KUKA KRL program: EPS_2_25252_SD5_A_20250910061729.src

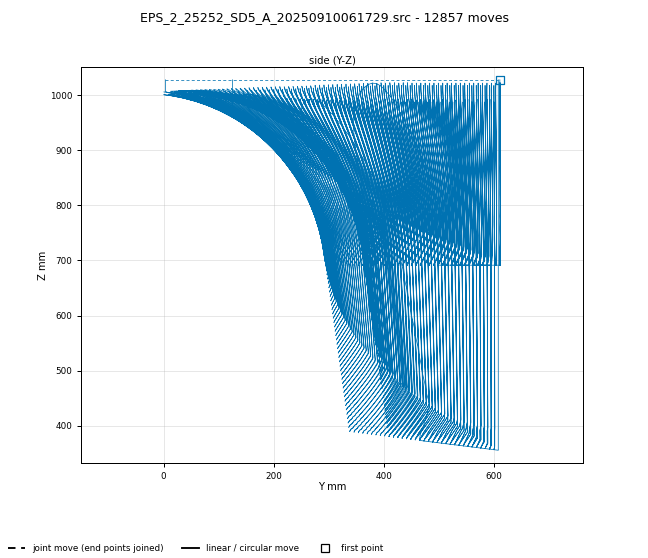
[picture p0: tool path of EPS_2_25252_SD5_A_20250910061729.src, 12857 of 12859 moves have a stored position in this frame; points joined in program order, loops and branches not executed]
&ACCESS RVP
&REL 4
&COMMENT QRS 19112012
&PARAM EDITMASK = *
DEF PART()
EXT BAS (BAS_COMMAND :IN,REAL :IN )
INT I
BAS (#INITMOV,0 )

;KUKA QRS Post kuka4.cps  Date:22-06-2017 !

File_ID=2833

QRS_PRE_INIT()

;Init var - Until changes are made in qrs_pre_init
Outlet_Square_prg=0
Inlet_1_Square_prg=0
Inlet_2_Square_prg=0
Inlet_3_Square_prg=0
Inlet_4_Square_prg=0
Inlet_5_Square_prg=0

Outlet_1={X 0.000, Y 400.000, Z 713.000, B 0.000, E1 0.000 }
Inlet_1={X 0.000, Y 400.000, Z 683.000, B 0.000, E1 212.000 }
Outlet_1_type=610
Inlet_1_type=610
;QRS#1=Sidecore dimensions
;QRS#2=600-24" Concrete
;QRS#3=600-24" Concrete
;QRS#4=
;QRS#5=
;QRS#6=
;QRS#7=
;QRS#8=
;QRS#9=S306-34L
;QRS#10=S306-34L
;QRS#11=
;QRS#12=
;QRS#13=
;QRS#14=
;QRS#15=
;QRS#16=1220x127x1372 4,5'
;QRS#17=EPS Height
;QRS#18=1018
;QRS#19=*
;QRS#20= UPDATED VERSION 22-06-2017
;QRS#21=*
Outlet_Square=0450
Inlet_1_Square=0450
Inlet_2_Square=0
Inlet_3_Square=0
Inlet_4_Square=0
Inlet_5_Square=0
Mill_Square=1
Outlet_Square_Prg=264
Inlet_1_Square_prg=264

QRS_INIT()

$ADVANCE=5

; T1
PTP {E1 178.273,E2 178.273}
PTP {X 0,Y 610.751,A -85,B 0,C 180,E1 178.273,E2 178.273,E3 0,E4 0,E5 0,E6 0}
QRS_SPEED_INIT()
LIN {X 0,Y 610.751,Z 1028,A -85,B 0,C 180,E1 178.273,E2 178.273,E3 0,E4 0,E5 0,E6 0} C_VEL
LIN {X 0,Y 610.751,Z 693.44,A -85,B 0,C 180,E1 178.273,E2 178.273} C_VEL
LIN {X 0,Y 610.777,Z 691.44,A -85,B 0,C 180,E1 178.46,E2 178.46} C_VEL
LIN {X 0,Y 611.879,Z 691.44,A -85,B 0,C 180,E1 181.167,E2 181.167} C_VEL
LIN {X 0,Y 611.804,Z 691.44,A -85,B 0,C 180,E1 188.197,E2 188.197} C_VEL
LIN {X 0,Y 611.819,Z 691.44,A -85,B 0,C 180,E1 195.354,E2 195.354} C_VEL
LIN {X 0,Y 611.767,Z 691.44,A -85,B 0,C 180,E1 202.769,E2 202.769} C_VEL
LIN {X 0,Y 611.74,Z 691.44,A -85,B 0,C 180,E1 210.614,E2 210.614} C_VEL
LIN {X 0,Y 610.579,Z 691.44,A -85,B 0,C 180,E1 217.262,E2 217.262} C_VEL
LIN {X 0,Y 611.716,Z 691.44,A -85,B 0,C 180,E1 219.161,E2 219.161} C_VEL
LIN {X 0,Y 610.312,Z 691.44,A -85,B 0,C 180,E1 222.361,E2 222.361} C_VEL
LIN {X 0,Y 610.625,Z 691.44,A -85,B 0,C 180,E1 225.583,E2 225.583} C_VEL
LIN {X 0,Y 611.712,Z 691.44,A -85,B 0,C 180,E1 227.764,E2 227.764} C_VEL
LIN {X 0,Y 611.693,Z 691.44,A -85,B 0,C 180,E1 235.933,E2 235.933} C_VEL
LIN {X 0,Y 611.734,Z 691.44,A -85,B 0,C 180,E1 236.287,E2 236.287} C_VEL
LIN {X 0,Y 611.056,Z 691.44,A -85,B 0,C 180,E1 236.42,E2 236.42} C_VEL
LIN {X 0,Y 610.433,Z 691.484,A -85,B 0,C 180,E1 236.481,E2 236.481} C_VEL
LIN {X 0,Y 611.412,Z 730.58,A -85,B 0,C 180,E1 237.083,E2 237.083} C_VEL
LIN {X 0,Y 611.517,Z 745.271,A -85,B 0,C 180,E1 237.336,E2 237.336} C_VEL
LIN {X 0,Y 611.325,Z 761.355,A -85,B 0,C 180,E1 237.681,E2 237.681} C_VEL
LIN {X 0,Y 611.672,Z 775.492,A -85,B 0,C 180,E1 238.087,E2 238.087} C_VEL
LIN {X 0,Y 611.736,Z 790.247,A -85,B 0,C 180,E1 238.57,E2 238.57} C_VEL
LIN {X 0,Y 611.693,Z 805.404,A -85,B 0,C 180,E1 239.145,E2 239.145} C_VEL
LIN {X 0,Y 611.448,Z 819.865,A -85,B 0,C 180,E1 239.763,E2 239.763} C_VEL
LIN {X 0,Y 611.625,Z 833.379,A -85,B 0,C 180,E1 240.435,E2 240.435} C_VEL
LIN {X 0,Y 611.599,Z 846.987,A -85,B 0,C 180,E1 241.179,E2 241.179} C_VEL
LIN {X 0,Y 611.634,Z 859.681,A -85,B 0,C 180,E1 241.947,E2 241.947} C_VEL
LIN {X 0,Y 611.641,Z 873.336,A -85,B 0,C 180,E1 242.859,E2 242.859} C_VEL
LIN {X 0,Y 611.572,Z 885.151,A -85,B 0,C 180,E1 243.716,E2 243.716} C_VEL
LIN {X 0,Y 611.333,Z 897.156,A -85,B 0,C 180,E1 244.659,E2 244.659} C_VEL
LIN {X 0,Y 611.276,Z 908.946,A -85,B 0,C 180,E1 245.678,E2 245.678} C_VEL
LIN {X 0,Y 611.472,Z 919.358,A -85,B 0,C 180,E1 246.662,E2 246.662} C_VEL
LIN {X 0,Y 611.734,Z 929.985,A -85,B 0,C 180,E1 247.752,E2 247.752} C_VEL
LIN {X 0,Y 611.445,Z 939.604,A -85,B 0,C 180,E1 248.799,E2 248.799} C_VEL
LIN {X 0,Y 611.088,Z 948.773,A -85,B 0,C 180,E1 249.876,E2 249.876} C_VEL
LIN {X 0,Y 611.074,Z 958.33,A -85,B 0,C 180,E1 251.115,E2 251.115} C_VEL
LIN {X 0,Y 611.399,Z 966.016,A -85,B 0,C 180,E1 252.202,E2 252.202} C_VEL
LIN {X 0,Y 611.821,Z 973.294,A -85,B 0,C 180,E1 253.324,E2 253.324} C_VEL
LIN {X 0,Y 611.107,Z 982.504,A -85,B 0,C 180,E1 254.862,E2 254.862} C_VEL
LIN {X 0,Y 610.739,Z 989.282,A -85,B 0,C 180,E1 256.129,E2 256.129} C_VEL
LIN {X 0,Y 610.875,Z 995.064,A -85,B 0,C 180,E1 257.336,E2 257.336} C_VEL
LIN {X 0,Y 611.566,Z 1001.374,A -85,B 0,C 180,E1 258.842,E2 258.842} C_VEL
LIN {X 0,Y 611.85,Z 1003.593,A -85,B 0,C 180,E1 259.441,E2 259.441} C_VEL
LIN {X 0,Y 611.525,Z 1005.813,A -85,B 0,C 180,E1 260.028,E2 260.028} C_VEL
LIN {X 0,Y 610.929,Z 1009.654,A -85,B 0,C 180,E1 261.203,E2 261.203} C_VEL
LIN {X 0,Y 610.672,Z 1012.99,A -85,B 0,C 180,E1 262.381,E2 262.381} C_VEL
LIN {X 0,Y 610.672,Z 1014.551,A -85,B 0,C 180,E1 262.97,E2 262.97} C_VEL
LIN {X 0,Y 611.06,Z 1017.122,A -85,B 0,C 180,E1 264.15,E2 264.15} C_VEL
LIN {X 0,Y 611.711,Z 1019.175,A -85,B 0,C 180,E1 265.329,E2 265.329} C_VEL
LIN {X 0,Y 611.37,Z 1020.807,A -85,B 0,C 180,E1 266.497,E2 266.497} C_VEL
LIN {X 0,Y 610.858,Z 1021.972,A -85,B 0,C 180,E1 267.634,E2 267.634} C_VEL
LIN {X 0,Y 610.688,Z 1022.778,A -85,B 0,C 180,E1 269.07,E2 269.07} C_VEL
LIN {X 0,Y 611.538,Z 1022.689,A -85,B 0,C 180,E1 271.17,E2 271.17} C_VEL
LIN {X 0,Y 611.319,Z 1021.671,A -85,B 0,C 180,E1 272.765,E2 272.765} C_VEL
LIN {X 0,Y 611.035,Z 1020.812,A -85,B 0,C 180,E1 273.51,E2 273.51} C_VEL
LIN {X 0,Y 610.805,Z 1019.195,A -85,B 0,C 180,E1 274.683,E2 274.683} C_VEL
LIN {X 0,Y 611.004,Z 1017.112,A -85,B 0,C 180,E1 275.855,E2 275.855} C_VEL
LIN {X 0,Y 611.55,Z 1014.528,A -85,B 0,C 180,E1 277.025,E2 277.025} C_VEL
LIN {X 0,Y 611.873,Z 1012.96,A -85,B 0,C 180,E1 277.609,E2 277.609} C_VEL
LIN {X 0,Y 611.24,Z 1009.637,A -85,B 0,C 180,E1 278.797,E2 278.797} C_VEL
LIN {X 0,Y 610.738,Z 1005.794,A -85,B 0,C 180,E1 279.99,E2 279.99} C_VEL
LIN {X 0,Y 610.738,Z 1000.148,A -85,B 0,C 180,E1 281.477,E2 281.477} C_VEL
LIN {X 0,Y 611.199,Z 995.041,A -85,B 0,C 180,E1 282.663,E2 282.663} C_VEL
LIN {X 0,Y 611.828,Z 989.347,A -85,B 0,C 180,E1 283.832,E2 283.832} C_VEL
LIN {X 0,Y 611.263,Z 982.265,A -85,B 0,C 180,E1 285.179,E2 285.179} C_VEL
LIN {X 0,Y 610.874,Z 973.74,A -85,B 0,C 180,E1 286.634,E2 286.634} C_VEL
LIN {X 0,Y 611.107,Z 964.917,A -85,B 0,C 180,E1 287.966,E2 287.966} C_VEL
LIN {X 0,Y 611.627,Z 956.005,A -85,B 0,C 180,E1 289.182,E2 289.182} C_VEL
LIN {X 0,Y 611.763,Z 951.156,A -85,B 0,C 180,E1 289.796,E2 289.796} C_VEL
LIN {X 0,Y 611.529,Z 944.982,A -85,B 0,C 180,E1 290.565,E2 290.565} C_VEL
LIN {X 0,Y 611.268,Z 937.362,A -85,B 0,C 180,E1 291.465,E2 291.465} C_VEL
LIN {X 0,Y 611.182,Z 926.924,A -85,B 0,C 180,E1 292.59,E2 292.59} C_VEL
LIN {X 0,Y 611.438,Z 916.307,A -85,B 0,C 180,E1 293.633,E2 293.633} C_VEL
LIN {X 0,Y 611.68,Z 905.115,A -85,B 0,C 180,E1 294.645,E2 294.645} C_VEL
LIN {X 0,Y 611.642,Z 894.627,A -85,B 0,C 180,E1 295.535,E2 295.535} C_VEL
LIN {X 0,Y 611.47,Z 882.904,A -85,B 0,C 180,E1 296.459,E2 296.459} C_VEL
LIN {X 0,Y 611.456,Z 869.528,A -85,B 0,C 180,E1 297.413,E2 297.413} C_VEL
LIN {X 0,Y 611.583,Z 857.645,A -85,B 0,C 180,E1 298.184,E2 298.184} C_VEL
LIN {X 0,Y 611.506,Z 843.831,A -85,B 0,C 180,E1 299.006,E2 299.006} C_VEL
LIN {X 0,Y 611.705,Z 829.667,A -85,B 0,C 180,E1 299.75,E2 299.75} C_VEL
LIN {X 0,Y 611.695,Z 816.022,A -85,B 0,C 180,E1 300.401,E2 300.401} C_VEL
LIN {X 0,Y 611.697,Z 800.989,A -85,B 0,C 180,E1 301.031,E2 301.031} C_VEL
LIN {X 0,Y 611.541,Z 786.837,A -85,B 0,C 180,E1 301.558,E2 301.558} C_VEL
LIN {X 0,Y 611.397,Z 780.445,A -85,B 0,C 180,E1 301.77,E2 301.77} C_VEL
LIN {X 0,Y 611.662,Z 771.874,A -85,B 0,C 180,E1 302.018,E2 302.018} C_VEL
LIN {X 0,Y 611.795,Z 756.357,A -85,B 0,C 180,E1 302.41,E2 302.41} C_VEL
LIN {X 0,Y 611.777,Z 742.708,A -85,B 0,C 180,E1 302.698,E2 302.698} C_VEL
LIN {X 0,Y 611.541,Z 723.406,A -85,B 0,C 180,E1 303.011,E2 303.011} C_VEL
LIN {X 0,Y 610.652,Z 696.32,A -85,B 0,C 180,E1 303.438,E2 303.438} C_VEL
LIN {X 0,Y 610.425,Z 691.44,A -85,B 0,C 180,E1 303.52,E2 303.52} C_VEL
LIN {X 0,Y 610.949,Z 691.44,A -85,B 0,C 180,E1 303.571,E2 303.571} C_VEL
LIN {X 0,Y 611.627,Z 691.44,A -85,B 0,C 180,E1 303.682,E2 303.682} C_VEL
LIN {X 0,Y 611.854,Z 691.44,A -85,B 0,C 180,E1 303.975,E2 303.975} C_VEL
LIN {X 0,Y 611.819,Z 691.44,A -85,B 0,C 180,E1 306.206,E2 306.206} C_VEL
LIN {X 0,Y 610.447,Z 691.44,A -85,B 0,C 180,E1 309.26,E2 309.26} C_VEL
LIN {X 0,Y 610.689,Z 691.44,A -85,B 0,C 180,E1 312.33,E2 312.33} C_VEL
LIN {X 0,Y 611.706,Z 691.44,A -85,B 0,C 180,E1 314.52,E2 314.52} C_VEL
LIN {X 0,Y 611.667,Z 691.44,A -85,B 0,C 180,E1 322.613,E2 322.613} C_VEL
LIN {X 0,Y 611.137,Z 691.44,A -85,B 0,C 180,E1 323.749,E2 323.749} C_VEL
LIN {X 0,Y 611.64,Z 691.44,A -85,B 0,C 180,E1 331.173,E2 331.173} C_VEL
LIN {X 0,Y 611.418,Z 691.44,A -85,B 0,C 180,E1 332.046,E2 332.046} C_VEL
LIN {X 0,Y 611.836,Z 691.44,A -85,B 0,C 180,E1 339.742,E2 339.742} C_VEL
LIN {X 0,Y 611.807,Z 691.44,A -85,B 0,C 180,E1 347.053,E2 347.053} C_VEL
LIN {X 0,Y 611.862,Z 691.44,A -85,B 0,C 180,E1 354.155,E2 354.155} C_VEL
LIN {X 0,Y 611.865,Z 691.44,A -85,B 0,C 180,E1 361.167,E2 361.167} C_VEL
LIN {X 0,Y 611.872,Z 691.44,A -85,B 0,C 180,E1 368.196,E2 368.196} C_VEL
LIN {X 0,Y 611.844,Z 691.44,A -85,B 0,C 180,E1 375.353,E2 375.353} C_VEL
LIN {X 0,Y 611.848,Z 691.44,A -85,B 0,C 180,E1 384.526,E2 384.526} C_VEL
LIN {X 0,Y 611.658,Z 691.44,A -85,B 0,C 180,E1 384.695,E2 384.695} C_VEL
LIN {X 0,Y 610.853,Z 691.44,A -85,B 0,C 180,E1 384.828,E2 384.828} C_VEL
LIN {X 0,Y 610.675,Z 693.966,A -85,B 0,C 180,E1 384.899,E2 384.899} C_VEL
LIN {X 0,Y 611.267,Z 713.813,A -85,B 0,C 180,E1 385.246,E2 385.246} C_VEL
LIN {X 0,Y 611.427,Z 721.576,A -85,B 0,C 180,E1 385.42,E2 385.42} C_VEL
LIN {X 0,Y 611.68,Z 731.96,A -85,B 0,C 180,E1 385.673,E2 385.673} C_VEL
LIN {X 0,Y 611.76,Z 746.114,A -85,B 0,C 180,E1 386.066,E2 386.066} C_VEL
LIN {X 0,Y 611.733,Z 760.823,A -85,B 0,C 180,E1 386.546,E2 386.546} C_VEL
LIN {X 0,Y 611.505,Z 775.533,A -85,B 0,C 180,E1 387.094,E2 387.094} C_VEL
LIN {X 0,Y 611.496,Z 780.73,A -85,B 0,C 180,E1 387.317,E2 387.317} C_VEL
LIN {X 0,Y 611.641,Z 790.77,A -85,B 0,C 180,E1 387.771,E2 387.771} C_VEL
LIN {X 0,Y 611.62,Z 803.533,A -85,B 0,C 180,E1 388.398,E2 388.398} C_VEL
LIN {X 0,Y 611.613,Z 815.956,A -85,B 0,C 180,E1 389.072,E2 389.072} C_VEL
LIN {X 0,Y 611.683,Z 830.386,A -85,B 0,C 180,E1 389.951,E2 389.951} C_VEL
LIN {X 0,Y 611.594,Z 842.995,A -85,B 0,C 180,E1 390.786,E2 390.786} C_VEL
LIN {X 0,Y 611.473,Z 854.821,A -85,B 0,C 180,E1 391.64,E2 391.64} C_VEL
LIN {X 0,Y 611.291,Z 867.28,A -85,B 0,C 180,E1 392.622,E2 392.622} C_VEL
LIN {X 0,Y 611.35,Z 878.197,A -85,B 0,C 180,E1 393.566,E2 393.566} C_VEL
LIN {X 0,Y 611.61,Z 889.208,A -85,B 0,C 180,E1 394.607,E2 394.607} C_VEL
LIN {X 0,Y 611.673,Z 898.184,A -85,B 0,C 180,E1 395.51,E2 395.51} C_VEL
LIN {X 0,Y 611.256,Z 908.83,A -85,B 0,C 180,E1 396.655,E2 396.655} C_VEL
LIN {X 0,Y 610.958,Z 918.775,A -85,B 0,C 180,E1 397.826,E2 397.826} C_VEL
LIN {X 0,Y 611.078,Z 927.661,A -85,B 0,C 180,E1 398.976,E2 398.976} C_VEL
LIN {X 0,Y 611.608,Z 937.24,A -85,B 0,C 180,E1 400.35,E2 400.35} C_VEL
LIN {X 0,Y 611.762,Z 942.057,A -85,B 0,C 180,E1 401.089,E2 401.089} C_VEL
LIN {X 0,Y 611.373,Z 947.337,A -85,B 0,C 180,E1 401.938,E2 401.938} C_VEL
LIN {X 0,Y 611.05,Z 951.437,A -85,B 0,C 180,E1 402.618,E2 402.618} C_VEL
LIN {X 0,Y 610.804,Z 959.535,A -85,B 0,C 180,E1 404.139,E2 404.139} C_VEL
LIN {X 0,Y 611.194,Z 966.057,A -85,B 0,C 180,E1 405.529,E2 405.529} C_VEL
LIN {X 0,Y 611.755,Z 970.815,A -85,B 0,C 180,E1 406.654,E2 406.654} C_VEL
LIN {X 0,Y 611.79,Z 972.216,A -85,B 0,C 180,E1 407.026,E2 407.026} C_VEL
LIN {X 0,Y 611.192,Z 976.094,A -85,B 0,C 180,E1 408.056,E2 408.056} C_VEL
LIN {X 0,Y 610.639,Z 980.184,A -85,B 0,C 180,E1 409.319,E2 409.319} C_VEL
LIN {X 0,Y 610.621,Z 984.118,A -85,B 0,C 180,E1 410.754,E2 410.754} C_VEL
LIN {X 0,Y 610.986,Z 986.189,A -85,B 0,C 180,E1 411.678,E2 411.678} C_VEL
LIN {X 0,Y 611.508,Z 988.084,A -85,B 0,C 180,E1 412.631,E2 412.631} C_VEL
LIN {X 0,Y 611.543,Z 989.989,A -85,B 0,C 180,E1 413.775,E2 413.775} C_VEL
LIN {X 0,Y 610.885,Z 991.668,A -85,B 0,C 180,E1 415.167,E2 415.167} C_VEL
LIN {X 0,Y 610.75,Z 992.718,A -85,B 0,C 180,E1 416.776,E2 416.776} C_VEL
LIN {X 0,Y 611.182,Z 992.972,A -85,B 0,C 180,E1 418.003,E2 418.003} C_VEL
LIN {X 0,Y 611.839,Z 992.593,A -85,B 0,C 180,E1 419.389,E2 419.389} C_VEL
LIN {X 0,Y 610.897,Z 991.017,A -85,B 0,C 180,E1 421.299,E2 421.299} C_VEL
LIN {X 0,Y 610.729,Z 990.169,A -85,B 0,C 180,E1 422.01,E2 422.01} C_VEL
LIN {X 0,Y 610.81,Z 988.415,A -85,B 0,C 180,E1 423.099,E2 423.099} C_VEL
LIN {X 0,Y 611.065,Z 986.959,A -85,B 0,C 180,E1 423.879,E2 423.879} C_VEL
LIN {X 0,Y 611.731,Z 984.138,A -85,B 0,C 180,E1 425.131,E2 425.131} C_VEL
LIN {X 0,Y 611.776,Z 982.892,A -85,B 0,C 180,E1 425.592,E2 425.592} C_VEL
LIN {X 0,Y 611.256,Z 980.295,A -85,B 0,C 180,E1 426.548,E2 426.548} C_VEL
LIN {X 0,Y 610.728,Z 975.416,A -85,B 0,C 180,E1 428.046,E2 428.046} C_VEL
LIN {X 0,Y 610.839,Z 970.323,A -85,B 0,C 180,E1 429.389,E2 429.389} C_VEL
LIN {X 0,Y 611.405,Z 964.84,A -85,B 0,C 180,E1 430.657,E2 430.657} C_VEL
LIN {X 0,Y 611.84,Z 960.265,A -85,B 0,C 180,E1 431.596,E2 431.596} C_VEL
LIN {X 0,Y 611.428,Z 955.618,A -85,B 0,C 180,E1 432.506,E2 432.506} C_VEL
LIN {X 0,Y 611.073,Z 950.639,A -85,B 0,C 180,E1 433.426,E2 433.426} C_VEL
LIN {X 0,Y 610.903,Z 943.532,A -85,B 0,C 180,E1 434.621,E2 434.621} C_VEL
LIN {X 0,Y 611.245,Z 935.024,A -85,B 0,C 180,E1 435.902,E2 435.902} C_VEL
LIN {X 0,Y 611.779,Z 925.47,A -85,B 0,C 180,E1 437.2,E2 437.2} C_VEL
LIN {X 0,Y 611.441,Z 916.141,A -85,B 0,C 180,E1 438.388,E2 438.388} C_VEL
LIN {X 0,Y 611.144,Z 907.369,A -85,B 0,C 180,E1 439.423,E2 439.423} C_VEL
LIN {X 0,Y 611.128,Z 897.783,A -85,B 0,C 180,E1 440.461,E2 440.461} C_VEL
LIN {X 0,Y 611.405,Z 887.269,A -85,B 0,C 180,E1 441.5,E2 441.5} C_VEL
LIN {X 0,Y 611.656,Z 875.889,A -85,B 0,C 180,E1 442.535,E2 442.535} C_VEL
LIN {X 0,Y 611.598,Z 863.723,A -85,B 0,C 180,E1 443.563,E2 443.563} C_VEL
LIN {X 0,Y 611.478,Z 852.503,A -85,B 0,C 180,E1 444.443,E2 444.443} C_VEL
LIN {X 0,Y 611.508,Z 840.182,A -85,B 0,C 180,E1 445.322,E2 445.322} C_VEL
LIN {X 0,Y 611.607,Z 826.174,A -85,B 0,C 180,E1 446.226,E2 446.226} C_VEL
LIN {X 0,Y 611.582,Z 817.202,A -85,B 0,C 180,E1 446.764,E2 446.764} C_VEL
LIN {X 0,Y 611.691,Z 800.766,A -85,B 0,C 180,E1 447.653,E2 447.653} C_VEL
LIN {X 0,Y 611.672,Z 786.231,A -85,B 0,C 180,E1 448.349,E2 448.349} C_VEL
LIN {X 0,Y 611.667,Z 771.537,A -85,B 0,C 180,E1 448.968,E2 448.968} C_VEL
LIN {X 0,Y 611.369,Z 756.142,A -85,B 0,C 180,E1 449.546,E2 449.546} C_VEL
LIN {X 0,Y 611.711,Z 741.221,A -85,B 0,C 180,E1 449.989,E2 449.989} C_VEL
LIN {X 0,Y 611.774,Z 726.511,A -85,B 0,C 180,E1 450.364,E2 450.364} C_VEL
LIN {X 0,Y 611.699,Z 711.57,A -85,B 0,C 180,E1 450.677,E2 450.677} C_VEL
LIN {X 0,Y 611.203,Z 694.049,A -85,B 0,C 180,E1 450.978,E2 450.978} C_VEL
LIN {X 0,Y 610.339,Z 691.44,A -85,B 0,C 180,E1 451.067,E2 451.067} C_VEL
LIN {X 0,Y 611.11,Z 691.44,A -85,B 0,C 180,E1 451.166,E2 451.166} C_VEL
LIN {X 0,Y 611.815,Z 691.44,A -85,B 0,C 180,E1 451.577,E2 451.577} C_VEL
LIN {X 0,Y 611.867,Z 691.44,A -85,B 0,C 180,E1 458.193,E2 458.193} C_VEL
LIN {X 0,Y 611.84,Z 691.44,A -85,B 0,C 180,E1 465.35,E2 465.35} C_VEL
LIN {X 0,Y 611.83,Z 691.44,A -85,B 0,C 180,E1 472.763,E2 472.763} C_VEL
LIN {X 0,Y 611.805,Z 691.44,A -85,B 0,C 180,E1 480.607,E2 480.607} C_VEL
LIN {X 0,Y 610.637,Z 691.44,A -85,B 0,C 180,E1 487.262,E2 487.262} C_VEL
LIN {X 0,Y 611.767,Z 691.44,A -85,B 0,C 180,E1 489.152,E2 489.152} C_VEL
LIN {X 0,Y 610.361,Z 691.44,A -85,B 0,C 180,E1 492.351,E2 492.351} C_VEL
LIN {X 0,Y 610.672,Z 691.44,A -85,B 0,C 180,E1 495.573,E2 495.573} C_VEL
LIN {X 0,Y 611.768,Z 691.44,A -85,B 0,C 180,E1 497.764,E2 497.764} C_VEL
LIN {X 0,Y 611.805,Z 691.44,A -85,B 0,C 180,E1 506.618,E2 506.618} C_VEL
LIN {X 0,Y 611.825,Z 691.44,A -85,B 0,C 180,E1 514.677,E2 514.677} C_VEL
LIN {X 0,Y 611.48,Z 691.44,A -85,B 0,C 180,E1 523.282,E2 523.282} C_VEL
LIN {X 0,Y 611.642,Z 691.44,A -85,B 0,C 180,E1 524.642,E2 524.642} C_VEL
LIN {X 0,Y 611.861,Z 691.44,A -85,B 0,C 180,E1 527.054,E2 527.054} C_VEL
LIN {X 0,Y 611.82,Z 691.44,A -85,B 0,C 180,E1 534.155,E2 534.155} C_VEL
LIN {X 0,Y 610.777,Z 691.44,A -85,B 0,C 180,E1 538.46,E2 538.46} C_VEL
LIN {X 0,Y 603.357,Z 691.44,A -85,B 0,C 180,E1 541.753,E2 541.753} C_VEL
LIN {X 0,Y 603.138,Z 691.44,A -85,B 0,C 180,E1 549.394,E2 549.394} C_VEL
LIN {X 0,Y 603.025,Z 691.44,A -85,B 0,C 180,E1 556.801,E2 556.801} C_VEL
LIN {X 0,Y 602.766,Z 691.44,A -85,B 0,C 180,E1 564.521,E2 564.521} C_VEL
LIN {X 0,Y 602.606,Z 691.44,A -85,B 0,C 180,E1 572.47,E2 572.47} C_VEL
LIN {X 0,Y 603.22,Z 691.44,A -85,B 0,C 180,E1 579.885,E2 579.885} C_VEL
LIN {X 0,Y 603.381,Z 691.44,A -85,B 0,C 180,E1 588.201,E2 588.201} C_VEL
LIN {X 0,Y 603.771,Z 692.564,A -85,B 0,C 180,E1 596.077,E2 596.077} C_VEL
LIN {X 0,Y 604.809,Z 776.8,A -85,B 0,C 180,E1 597.724,E2 597.724} C_VEL
LIN {X 0,Y 604.426,Z 842.228,A -85,B 0,C 180,E1 600.533,E2 600.533} C_VEL
LIN {X 0,Y 603.772,Z 901.573,A -85,B 0,C 180,E1 604.703,E2 604.703} C_VEL
LIN {X 0,Y 603.279,Z 950,A -85,B 0,C 180,E1 609.763,E2 609.763} C_VEL
LIN {X 0,Y 603.004,Z 985.703,A -85,B 0,C 180,E1 615.257,E2 615.257} C_VEL
LIN {X 0,Y 603.039,Z 1009.219,A -85,B 0,C 180,E1 620.95,E2 620.95} C_VEL
LIN {X 0,Y 603.404,Z 1020.765,A -85,B 0,C 180,E1 626.394,E2 626.394} C_VEL
LIN {X 0,Y 603.378,Z 1022.149,A -85,B 0,C 180,E1 632.161,E2 632.161} C_VEL
LIN {X 0,Y 603.3,Z 1010.38,A -85,B 0,C 180,E1 638.68,E2 638.68} C_VEL
LIN {X 0,Y 603.37,Z 983.787,A -85,B 0,C 180,E1 645.095,E2 645.095} C_VEL
LIN {X 0,Y 603.641,Z 943.762,A -85,B 0,C 180,E1 650.992,E2 650.992} C_VEL
LIN {X 0,Y 604.094,Z 892.096,A -85,B 0,C 180,E1 656.08,E2 656.08} C_VEL
LIN {X 0,Y 604.609,Z 831.093,A -85,B 0,C 180,E1 660.065,E2 660.065} C_VEL
LIN {X 0,Y 604.94,Z 766.019,A -85,B 0,C 180,E1 662.576,E2 662.576} C_VEL
LIN {X 0,Y 603.83,Z 691.44,A -85,B 0,C 180,E1 663.957,E2 663.957} C_VEL
LIN {X 0,Y 603.526,Z 691.44,A -85,B 0,C 180,E1 674.26,E2 674.26} C_VEL
LIN {X 0,Y 603.113,Z 691.44,A -85,B 0,C 180,E1 683.78,E2 683.78} C_VEL
LIN {X 0,Y 603.275,Z 691.44,A -85,B 0,C 180,E1 692.291,E2 692.291} C_VEL
LIN {X 0,Y 602.86,Z 691.44,A -85,B 0,C 180,E1 701.682,E2 701.682} C_VEL
LIN {X 0,Y 602.87,Z 691.44,A -85,B 0,C 180,E1 709.137,E2 709.137} C_VEL
LIN {X 0,Y 602.867,Z 691.44,A -85,B 0,C 180,E1 716.409,E2 716.409} C_VEL
LIN {X 0,Y 602.825,Z 691.44,A -85,B 0,C 180,E1 723.624,E2 723.624} C_VEL
LIN {X 0,Y 603.211,Z 691.44,A -85,B 0,C 180,E1 729.426,E2 729.426} C_VEL
LIN {X 0,Y 602.794,Z 691.44,A -85,B 0,C 180,E1 736.843,E2 736.843} C_VEL
LIN {X 0,Y 603.921,Z 692.809,A -85,B 0,C 180,E1 744.465,E2 744.465} C_VEL
LIN {X 0,Y 604.795,Z 761.917,A -85,B 0,C 180,E1 746.185,E2 746.185} C_VEL
LIN {X 0,Y 604.399,Z 826.363,A -85,B 0,C 180,E1 749.327,E2 749.327} C_VEL
LIN {X 0,Y 603.824,Z 884.069,A -85,B 0,C 180,E1 753.795,E2 753.795} C_VEL
LIN {X 0,Y 603.31,Z 931.095,A -85,B 0,C 180,E1 759.208,E2 759.208} C_VEL
LIN {X 0,Y 603.126,Z 965.376,A -85,B 0,C 180,E1 765.197,E2 765.197} C_VEL
LIN {X 0,Y 602.701,Z 984.89,A -85,B 0,C 180,E1 770.988,E2 770.988} C_VEL
LIN {X 0,Y 602.841,Z 991.945,A -85,B 0,C 180,E1 775.5,E2 775.5} C_VEL
LIN {X 0,Y 603.161,Z 991.796,A -85,B 0,C 180,E1 780.619,E2 780.619} C_VEL
LIN {X 0,Y 603.195,Z 980.214,A -85,B 0,C 180,E1 786.69,E2 786.69} C_VEL
LIN {X 0,Y 603.365,Z 955.054,A -85,B 0,C 180,E1 792.811,E2 792.811} C_VEL
LIN {X 0,Y 603.624,Z 916.839,A -85,B 0,C 180,E1 798.581,E2 798.581} C_VEL
LIN {X 0,Y 604.089,Z 865.279,A -85,B 0,C 180,E1 803.781,E2 803.781} C_VEL
LIN {X 0,Y 604.551,Z 804.452,A -85,B 0,C 180,E1 807.843,E2 807.843} C_VEL
LIN {X 0,Y 604.889,Z 740.829,A -85,B 0,C 180,E1 810.405,E2 810.405} C_VEL
LIN {X 0,Y 603.804,Z 691.44,A -85,B 0,C 180,E1 811.621,E2 811.621} C_VEL
LIN {X 0,Y 603.212,Z 691.44,A -85,B 0,C 180,E1 819.413,E2 819.413} C_VEL
LIN {X 0,Y 603.036,Z 691.44,A -85,B 0,C 180,E1 826.823,E2 826.823} C_VEL
LIN {X 0,Y 602.825,Z 691.44,A -85,B 0,C 180,E1 834.544,E2 834.544} C_VEL
LIN {X 0,Y 602.661,Z 691.44,A -85,B 0,C 180,E1 842.471,E2 842.471} C_VEL
LIN {X 0,Y 603.27,Z 691.44,A -85,B 0,C 180,E1 849.903,E2 849.903} C_VEL
LIN {X 0,Y 603.418,Z 691.44,A -85,B 0,C 180,E1 858.195,E2 858.195} C_VEL
LIN {X 0,Y 603.258,Z 691.44,A -85,B 0,C 180,E1 867.433,E2 867.433} C_VEL
LIN {X 0,Y 603.206,Z 691.44,A -85,B 0,C 180,E1 875.461,E2 875.461} C_VEL
LIN {X 0,Y 603.686,Z 691.44,A -85,B 0,C 180,E1 886.17,E2 886.17} C_VEL
LIN {X 0,Y 603.367,Z 691.44,A -85,B 0,C 180,E1 894.934,E2 894.934} C_VEL
LIN {X 0,Y 603.357,Z 691.44,A -85,B 0,C 180,E1 901.753,E2 901.753} C_VEL
LIN {X 0,Y 594.729,Z 691.44,A -85,B 0,C 180,E1 905.047,E2 905.047} C_VEL
LIN {X 0,Y 594.681,Z 691.44,A -85,B 0,C 180,E1 911.014,E2 911.014} C_VEL
LIN {X 0,Y 594.932,Z 691.44,A -85,B 0,C 180,E1 917.037,E2 917.037} C_VEL
LIN {X 0,Y 594.592,Z 691.44,A -85,B 0,C 180,E1 925.03,E2 925.03} C_VEL
LIN {X 0,Y 595.111,Z 691.44,A -85,B 0,C 180,E1 931.49,E2 931.49} C_VEL
LIN {X 0,Y 594.615,Z 691.44,A -85,B 0,C 180,E1 941.156,E2 941.156} C_VEL
LIN {X 0,Y 594.717,Z 691.44,A -85,B 0,C 180,E1 949.404,E2 949.404} C_VEL
LIN {X 0,Y 595.531,Z 692.902,A -85,B 0,C 180,E1 955.546,E2 955.546} C_VEL
LIN {X 0,Y 597.95,Z 779.177,A -85,B 0,C 180,E1 957.386,E2 957.386} C_VEL
LIN {X 0,Y 597.262,Z 843.929,A -85,B 0,C 180,E1 960.238,E2 960.238} C_VEL
LIN {X 0,Y 596.216,Z 903.932,A -85,B 0,C 180,E1 964.567,E2 964.567} C_VEL
LIN {X 0,Y 595.471,Z 951.478,A -85,B 0,C 180,E1 969.681,E2 969.681} C_VEL
LIN {X 0,Y 595.078,Z 986.256,A -85,B 0,C 180,E1 975.162,E2 975.162} C_VEL
LIN {X 0,Y 594.979,Z 1010.375,A -85,B 0,C 180,E1 981.196,E2 981.196} C_VEL
LIN {X 0,Y 595.416,Z 1020.765,A -85,B 0,C 180,E1 986.346,E2 986.346} C_VEL
LIN {X 0,Y 595.363,Z 1022.149,A -85,B 0,C 180,E1 992.191,E2 992.191} C_VEL
LIN {X 0,Y 595.255,Z 1010.379,A -85,B 0,C 180,E1 998.798,E2 998.798} C_VEL
LIN {X 0,Y 595.435,Z 984.424,A -85,B 0,C 180,E1 1005.179,E2 1005.179} C_VEL
LIN {X 0,Y 595.87,Z 945.379,A -85,B 0,C 180,E1 1011.084,E2 1011.084} C_VEL
LIN {X 0,Y 596.619,Z 893.819,A -85,B 0,C 180,E1 1016.292,E2 1016.292} C_VEL
LIN {X 0,Y 597.462,Z 833.473,A -85,B 0,C 180,E1 1020.333,E2 1020.333} C_VEL
LIN {X 0,Y 598.096,Z 769.327,A -85,B 0,C 180,E1 1022.905,E2 1022.905} C_VEL
LIN {X 0,Y 595.783,Z 691.44,A -85,B 0,C 180,E1 1024.493,E2 1024.493} C_VEL
LIN {X 0,Y 594.966,Z 691.44,A -85,B 0,C 180,E1 1035.494,E2 1035.494} C_VEL
LIN {X 0,Y 595.188,Z 691.44,A -85,B 0,C 180,E1 1043.433,E2 1043.433} C_VEL
LIN {X 0,Y 595.224,Z 691.44,A -85,B 0,C 180,E1 1051.883,E2 1051.883} C_VEL
LIN {X 0,Y 594.944,Z 691.44,A -85,B 0,C 180,E1 1061.429,E2 1061.429} C_VEL
LIN {X 0,Y 594.886,Z 691.44,A -85,B 0,C 180,E1 1069.157,E2 1069.157} C_VEL
LIN {X 0,Y 594.877,Z 691.44,A -85,B 0,C 180,E1 1076.361,E2 1076.361} C_VEL
LIN {X 0,Y 594.815,Z 691.44,A -85,B 0,C 180,E1 1083.673,E2 1083.673} C_VEL
LIN {X 0,Y 594.787,Z 691.44,A -85,B 0,C 180,E1 1090.792,E2 1090.792} C_VEL
LIN {X 0,Y 594.669,Z 691.44,A -85,B 0,C 180,E1 1097.08,E2 1097.08} C_VEL
LIN {X 0,Y 595.613,Z 693.374,A -85,B 0,C 180,E1 1103.942,E2 1103.942} C_VEL
LIN {X 0,Y 597.873,Z 763.831,A -85,B 0,C 180,E1 1105.847,E2 1105.847} C_VEL
LIN {X 0,Y 597.146,Z 827.614,A -85,B 0,C 180,E1 1109.024,E2 1109.024} C_VEL
LIN {X 0,Y 596.184,Z 885.145,A -85,B 0,C 180,E1 1113.567,E2 1113.567} C_VEL
LIN {X 0,Y 595.462,Z 932.097,A -85,B 0,C 180,E1 1119.095,E2 1119.095} C_VEL
LIN {X 0,Y 595.157,Z 966.068,A -85,B 0,C 180,E1 1125.189,E2 1125.189} C_VEL
LIN {X 0,Y 594.837,Z 985.785,A -85,B 0,C 180,E1 1131.314,E2 1131.314} C_VEL
LIN {X 0,Y 594.814,Z 992.727,A -85,B 0,C 180,E1 1136.734,E2 1136.734} C_VEL
LIN {X 0,Y 594.793,Z 990.51,A -85,B 0,C 180,E1 1141.835,E2 1141.835} C_VEL
LIN {X 0,Y 594.92,Z 978.055,A -85,B 0,C 180,E1 1147.504,E2 1147.504} C_VEL
LIN {X 0,Y 595.287,Z 953.4,A -85,B 0,C 180,E1 1153.334,E2 1153.334} C_VEL
LIN {X 0,Y 595.72,Z 914.329,A -85,B 0,C 180,E1 1159.172,E2 1159.172} C_VEL
LIN {X 0,Y 596.605,Z 862.605,A -85,B 0,C 180,E1 1164.347,E2 1164.347} C_VEL
LIN {X 0,Y 597.467,Z 802.103,A -85,B 0,C 180,E1 1168.363,E2 1168.363} C_VEL
LIN {X 0,Y 598.146,Z 738.602,A -85,B 0,C 180,E1 1170.878,E2 1170.878} C_VEL
LIN {X 0,Y 595.949,Z 693.68,A -85,B 0,C 180,E1 1171.942,E2 1171.942} C_VEL
LIN {X 0,Y 595.476,Z 691.44,A -85,B 0,C 180,E1 1172.192,E2 1172.192} C_VEL
LIN {X 0,Y 595.152,Z 691.44,A -85,B 0,C 180,E1 1179.541,E2 1179.541} C_VEL
LIN {X 0,Y 594.944,Z 691.44,A -85,B 0,C 180,E1 1187.059,E2 1187.059} C_VEL
LIN {X 0,Y 594.662,Z 691.44,A -85,B 0,C 180,E1 1195.036,E2 1195.036} C_VEL
LIN {X 0,Y 595.189,Z 691.44,A -85,B 0,C 180,E1 1201.514,E2 1201.514} C_VEL
LIN {X 0,Y 594.682,Z 691.44,A -85,B 0,C 180,E1 1211.155,E2 1211.155} C_VEL
LIN {X 0,Y 594.68,Z 691.44,A -85,B 0,C 180,E1 1219.392,E2 1219.392} C_VEL
LIN {X 0,Y 594.771,Z 691.44,A -85,B 0,C 180,E1 1228.45,E2 1228.45} C_VEL
LIN {X 0,Y 594.514,Z 691.44,A -85,B 0,C 180,E1 1236.68,E2 1236.68} C_VEL
LIN {X 0,Y 595.66,Z 691.44,A -85,B 0,C 180,E1 1245.979,E2 1245.979} C_VEL
LIN {X 0,Y 595.381,Z 691.44,A -85,B 0,C 180,E1 1254.866,E2 1254.866} C_VEL
LIN {X 0,Y 595.311,Z 691.44,A -85,B 0,C 180,E1 1262.174,E2 1262.174} C_VEL
LIN {X 0,Y 594.729,Z 691.44,A -85,B 0,C 180,E1 1265.047,E2 1265.047} C_VEL
LIN {X 0,Y 587.442,Z 691.44,A -85,B 0,C 180,E1 1268.414,E2 1268.414} C_VEL
LIN {X 0,Y 586.843,Z 691.44,A -85,B 0,C 180,E1 1277.279,E2 1277.279} C_VEL
LIN {X 0,Y 586.537,Z 691.44,A -85,B 0,C 180,E1 1285.246,E2 1285.246} C_VEL
LIN {X 0,Y 586.479,Z 691.44,A -85,B 0,C 180,E1 1292.755,E2 1292.755} C_VEL
LIN {X 0,Y 586.58,Z 691.44,A -85,B 0,C 180,E1 1301.244,E2 1301.244} C_VEL
LIN {X 0,Y 587.051,Z 691.44,A -85,B 0,C 180,E1 1308.76,E2 1308.76} C_VEL
LIN {X 0,Y 587.268,Z 693.224,A -85,B 0,C 180,E1 1314.996,E2 1314.996} C_VEL
LIN {X 0,Y 590.806,Z 705.86,A -85,B 0,C 180,E1 1315.419,E2 1315.419} C_VEL
LIN {X 0,Y 591.127,Z 781.225,A -85,B 0,C 180,E1 1317.03,E2 1317.03} C_VEL
LIN {X 0,Y 590.116,Z 844.989,A -85,B 0,C 180,E1 1319.901,E2 1319.901} C_VEL
LIN {X 0,Y 588.713,Z 903.933,A -85,B 0,C 180,E1 1324.219,E2 1324.219} C_VEL
LIN {X 0,Y 587.669,Z 952.956,A -85,B 0,C 180,E1 1329.596,E2 1329.596} C_VEL
LIN {X 0,Y 587.123,Z 987.672,A -85,B 0,C 180,E1 1335.231,E2 1335.231} C_VEL
LIN {X 0,Y 587.026,Z 1010.375,A -85,B 0,C 180,E1 1341.076,E2 1341.076} C_VEL
LIN {X 0,Y 587.424,Z 1020.765,A -85,B 0,C 180,E1 1346.296,E2 1346.296} C_VEL
LIN {X 0,Y 587.349,Z 1022.149,A -85,B 0,C 180,E1 1352.22,E2 1352.22} C_VEL
LIN {X 0,Y 587.22,Z 1010.379,A -85,B 0,C 180,E1 1358.92,E2 1358.92} C_VEL
LIN {X 0,Y 587.435,Z 984.429,A -85,B 0,C 180,E1 1365.39,E2 1365.39} C_VEL
LIN {X 0,Y 588.112,Z 946.068,A -85,B 0,C 180,E1 1371.291,E2 1371.291} C_VEL
LIN {X 0,Y 589.149,Z 894.979,A -85,B 0,C 180,E1 1376.556,E2 1376.556} C_VEL
LIN {X 0,Y 590.399,Z 833.731,A -85,B 0,C 180,E1 1380.72,E2 1380.72} C_VEL
LIN {X 0,Y 591.338,Z 769.761,A -85,B 0,C 180,E1 1383.317,E2 1383.317} C_VEL
LIN {X 0,Y 588.991,Z 695.701,A -85,B 0,C 180,E1 1384.85,E2 1384.85} C_VEL
LIN {X 0,Y 587.701,Z 691.44,A -85,B 0,C 180,E1 1385.101,E2 1385.101} C_VEL
LIN {X 0,Y 587.029,Z 691.44,A -85,B 0,C 180,E1 1395.31,E2 1395.31} C_VEL
LIN {X 0,Y 586.67,Z 691.44,A -85,B 0,C 180,E1 1404.57,E2 1404.57} C_VEL
LIN {X 0,Y 586.736,Z 691.44,A -85,B 0,C 180,E1 1413.167,E2 1413.167} C_VEL
LIN {X 0,Y 586.996,Z 691.44,A -85,B 0,C 180,E1 1421.168,E2 1421.168} C_VEL
LIN {X 0,Y 586.96,Z 691.44,A -85,B 0,C 180,E1 1428.839,E2 1428.839} C_VEL
LIN {X 0,Y 586.888,Z 691.44,A -85,B 0,C 180,E1 1436.312,E2 1436.312} C_VEL
LIN {X 0,Y 586.807,Z 691.44,A -85,B 0,C 180,E1 1443.723,E2 1443.723} C_VEL
LIN {X 0,Y 587.123,Z 691.44,A -85,B 0,C 180,E1 1449.687,E2 1449.687} C_VEL
LIN {X 0,Y 586.535,Z 691.44,A -85,B 0,C 180,E1 1457.324,E2 1457.324} C_VEL
LIN {X 0,Y 587.182,Z 693.271,A -85,B 0,C 180,E1 1463.384,E2 1463.384} C_VEL
LIN {X 0,Y 590.961,Z 708.011,A -85,B 0,C 180,E1 1463.869,E2 1463.869} C_VEL
LIN {X 0,Y 590.701,Z 776.264,A -85,B 0,C 180,E1 1465.913,E2 1465.913} C_VEL
LIN {X 0,Y 589.708,Z 838.762,A -85,B 0,C 180,E1 1469.388,E2 1469.388} C_VEL
LIN {X 0,Y 588.615,Z 894.434,A -85,B 0,C 180,E1 1474.185,E2 1474.185} C_VEL
LIN {X 0,Y 587.846,Z 938.369,A -85,B 0,C 180,E1 1479.792,E2 1479.792} C_VEL
LIN {X 0,Y 587.649,Z 971.033,A -85,B 0,C 180,E1 1486.243,E2 1486.243} C_VEL
LIN {X 0,Y 587.442,Z 988.452,A -85,B 0,C 180,E1 1492.621,E2 1492.621} C_VEL
LIN {X 0,Y 587.152,Z 992.996,A -85,B 0,C 180,E1 1498.005,E2 1498.005} C_VEL
LIN {X 0,Y 587.513,Z 985.588,A -85,B 0,C 180,E1 1504.774,E2 1504.774} C_VEL
LIN {X 0,Y 587.865,Z 963.038,A -85,B 0,C 180,E1 1511.565,E2 1511.565} C_VEL
LIN {X 0,Y 588.196,Z 926.26,A -85,B 0,C 180,E1 1517.9,E2 1517.9} C_VEL
LIN {X 0,Y 588.981,Z 877.127,A -85,B 0,C 180,E1 1523.435,E2 1523.435} C_VEL
LIN {X 0,Y 590.053,Z 817.835,A -85,B 0,C 180,E1 1527.882,E2 1527.882} C_VEL
LIN {X 0,Y 590.996,Z 753.033,A -85,B 0,C 180,E1 1530.874,E2 1530.874} C_VEL
LIN {X 0,Y 589.49,Z 696.777,A -85,B 0,C 180,E1 1532.321,E2 1532.321} C_VEL
LIN {X 0,Y 587.299,Z 691.44,A -85,B 0,C 180,E1 1532.593,E2 1532.593} C_VEL
LIN {X 0,Y 587.125,Z 691.44,A -85,B 0,C 180,E1 1539.673,E2 1539.673} C_VEL
LIN {X 0,Y 586.862,Z 691.44,A -85,B 0,C 180,E1 1547.301,E2 1547.301} C_VEL
LIN {X 0,Y 586.605,Z 691.44,A -85,B 0,C 180,E1 1555.27,E2 1555.27} C_VEL
LIN {X 0,Y 586.551,Z 691.44,A -85,B 0,C 180,E1 1562.757,E2 1562.757} C_VEL
LIN {X 0,Y 586.642,Z 691.44,A -85,B 0,C 180,E1 1571.275,E2 1571.275} C_VEL
LIN {X 0,Y 587.029,Z 691.44,A -85,B 0,C 180,E1 1578.749,E2 1578.749} C_VEL
LIN {X 0,Y 586.837,Z 691.44,A -85,B 0,C 180,E1 1587.974,E2 1587.974} C_VEL
LIN {X 0,Y 586.488,Z 691.44,A -85,B 0,C 180,E1 1596.723,E2 1596.723} C_VEL
LIN {X 0,Y 587.629,Z 691.44,A -85,B 0,C 180,E1 1605.784,E2 1605.784} C_VEL
LIN {X 0,Y 587.373,Z 691.44,A -85,B 0,C 180,E1 1614.796,E2 1614.796} C_VEL
LIN {X 0,Y 587.29,Z 691.44,A -85,B 0,C 180,E1 1622.204,E2 1622.204} C_VEL
LIN {X 0,Y 587.442,Z 691.44,A -85,B 0,C 180,E1 1628.414,E2 1628.414} C_VEL
LIN {X 0,Y 578.649,Z 691.44,A -85,B 0,C 180,E1 1631.8,E2 1631.8} C_VEL
LIN {X 0,Y 578.553,Z 691.44,A -85,B 0,C 180,E1 1639.117,E2 1639.117} C_VEL
LIN {X 0,Y 578.455,Z 691.44,A -85,B 0,C 180,E1 1645.625,E2 1645.625} C_VEL
LIN {X 0,Y 578.577,Z 691.44,A -85,B 0,C 180,E1 1652.498,E2 1652.498} C_VEL
LIN {X 0,Y 578.465,Z 691.44,A -85,B 0,C 180,E1 1661.608,E2 1661.608} C_VEL
LIN {X 0,Y 578.511,Z 691.44,A -85,B 0,C 180,E1 1670.005,E2 1670.005} C_VEL
LIN {X 0,Y 579.011,Z 693.366,A -85,B 0,C 180,E1 1674.424,E2 1674.424} C_VEL
LIN {X 0,Y 584.248,Z 707.736,A -85,B 0,C 180,E1 1675.002,E2 1675.002} C_VEL
LIN {X 0,Y 584.326,Z 783.331,A -85,B 0,C 180,E1 1676.668,E2 1676.668} C_VEL
LIN {X 0,Y 582.949,Z 846.458,A -85,B 0,C 180,E1 1679.585,E2 1679.585} C_VEL
LIN {X 0,Y 581.182,Z 906.683,A -85,B 0,C 180,E1 1684.11,E2 1684.11} C_VEL
LIN {X 0,Y 579.852,Z 954.526,A -85,B 0,C 180,E1 1689.521,E2 1689.521} C_VEL
LIN {X 0,Y 579.175,Z 988.546,A -85,B 0,C 180,E1 1695.197,E2 1695.197} C_VEL
LIN {X 0,Y 579.069,Z 1010.374,A -85,B 0,C 180,E1 1700.952,E2 1700.952} C_VEL
LIN {X 0,Y 579.433,Z 1020.765,A -85,B 0,C 180,E1 1706.245,E2 1706.245} C_VEL
LIN {X 0,Y 579.345,Z 1022.149,A -85,B 0,C 180,E1 1712.251,E2 1712.251} C_VEL
LIN {X 0,Y 579.208,Z 1010.379,A -85,B 0,C 180,E1 1719.044,E2 1719.044} C_VEL
LIN {X 0,Y 579.514,Z 985.603,A -85,B 0,C 180,E1 1725.375,E2 1725.375} C_VEL
LIN {X 0,Y 580.308,Z 946.133,A -85,B 0,C 180,E1 1731.583,E2 1731.583} C_VEL
LIN {X 0,Y 581.691,Z 894.352,A -85,B 0,C 180,E1 1736.977,E2 1736.977} C_VEL
LIN {X 0,Y 583.362,Z 833.21,A -85,B 0,C 180,E1 1741.161,E2 1741.161} C_VEL
LIN {X 0,Y 584.625,Z 769.763,A -85,B 0,C 180,E1 1743.751,E2 1743.751} C_VEL
LIN {X 0,Y 582.42,Z 698.389,A -85,B 0,C 180,E1 1745.262,E2 1745.262} C_VEL
LIN {X 0,Y 579.552,Z 691.44,A -85,B 0,C 180,E1 1745.703,E2 1745.703} C_VEL
LIN {X 0,Y 578.672,Z 691.44,A -85,B 0,C 180,E1 1756.153,E2 1756.153} C_VEL
LIN {X 0,Y 578.756,Z 691.44,A -85,B 0,C 180,E1 1763.876,E2 1763.876} C_VEL
LIN {X 0,Y 578.814,Z 691.44,A -85,B 0,C 180,E1 1772.715,E2 1772.715} C_VEL
LIN {X 0,Y 579.082,Z 691.44,A -85,B 0,C 180,E1 1780.901,E2 1780.901} C_VEL
LIN {X 0,Y 578.787,Z 691.44,A -85,B 0,C 180,E1 1789.497,E2 1789.497} C_VEL
LIN {X 0,Y 578.923,Z 691.44,A -85,B 0,C 180,E1 1796.261,E2 1796.261} C_VEL
LIN {X 0,Y 578.829,Z 691.44,A -85,B 0,C 180,E1 1803.775,E2 1803.775} C_VEL
LIN {X 0,Y 578.879,Z 691.44,A -85,B 0,C 180,E1 1810.552,E2 1810.552} C_VEL
LIN {X 0,Y 578.444,Z 691.44,A -85,B 0,C 180,E1 1817.574,E2 1817.574} C_VEL
LIN {X 0,Y 578.79,Z 692.961,A -85,B 0,C 180,E1 1822.805,E2 1822.805} C_VEL
LIN {X 0,Y 584.314,Z 707.838,A -85,B 0,C 180,E1 1823.424,E2 1823.424} C_VEL
LIN {X 0,Y 583.858,Z 775.765,A -85,B 0,C 180,E1 1825.469,E2 1825.469} C_VEL
LIN {X 0,Y 582.442,Z 838.78,A -85,B 0,C 180,E1 1828.999,E2 1828.999} C_VEL
LIN {X 0,Y 580.961,Z 893.965,A -85,B 0,C 180,E1 1833.802,E2 1833.802} C_VEL
LIN {X 0,Y 579.943,Z 938.959,A -85,B 0,C 180,E1 1839.63,E2 1839.63} C_VEL
LIN {X 0,Y 579.621,Z 970.986,A -85,B 0,C 180,E1 1846.066,E2 1846.066} C_VEL
LIN {X 0,Y 579.414,Z 989.231,A -85,B 0,C 180,E1 1853.031,E2 1853.031} C_VEL
LIN {X 0,Y 579.247,Z 992.714,A -85,B 0,C 180,E1 1859.278,E2 1859.278} C_VEL
LIN {X 0,Y 579.393,Z 982.214,A -85,B 0,C 180,E1 1866.293,E2 1866.293} C_VEL
LIN {X 0,Y 579.559,Z 957.747,A -85,B 0,C 180,E1 1872.907,E2 1872.907} C_VEL
LIN {X 0,Y 580.22,Z 920.078,A -85,B 0,C 180,E1 1879.025,E2 1879.025} C_VEL
LIN {X 0,Y 581.595,Z 869.49,A -85,B 0,C 180,E1 1884.481,E2 1884.481} C_VEL
LIN {X 0,Y 583.134,Z 810.794,A -85,B 0,C 180,E1 1888.696,E2 1888.696} C_VEL
LIN {X 0,Y 584.508,Z 746.343,A -85,B 0,C 180,E1 1891.514,E2 1891.514} C_VEL
LIN {X 0,Y 583.049,Z 700.53,A -85,B 0,C 180,E1 1892.697,E2 1892.697} C_VEL
LIN {X 0,Y 579.086,Z 691.44,A -85,B 0,C 180,E1 1893.194,E2 1893.194} C_VEL
LIN {X 0,Y 578.861,Z 691.44,A -85,B 0,C 180,E1 1900.519,E2 1900.519} C_VEL
LIN {X 0,Y 578.816,Z 691.44,A -85,B 0,C 180,E1 1907.55,E2 1907.55} C_VEL
LIN {X 0,Y 578.531,Z 691.44,A -85,B 0,C 180,E1 1915.648,E2 1915.648} C_VEL
LIN {X 0,Y 578.648,Z 691.44,A -85,B 0,C 180,E1 1922.524,E2 1922.524} C_VEL
LIN {X 0,Y 578.553,Z 691.44,A -85,B 0,C 180,E1 1931.609,E2 1931.609} C_VEL
LIN {X 0,Y 578.412,Z 691.44,A -85,B 0,C 180,E1 1939.987,E2 1939.987} C_VEL
LIN {X 0,Y 578.661,Z 691.44,A -85,B 0,C 180,E1 1948.469,E2 1948.469} C_VEL
LIN {X 0,Y 578.723,Z 691.44,A -85,B 0,C 180,E1 1956.005,E2 1956.005} C_VEL
LIN {X 0,Y 579.63,Z 691.44,A -85,B 0,C 180,E1 1965.583,E2 1965.583} C_VEL
LIN {X 0,Y 579.373,Z 691.44,A -85,B 0,C 180,E1 1974.724,E2 1974.724} C_VEL
LIN {X 0,Y 579.299,Z 691.44,A -85,B 0,C 180,E1 1982.234,E2 1982.234} C_VEL
LIN {X 0,Y 578.796,Z 691.44,A -85,B 0,C 180,E1 1990.5,E2 1990.5} C_VEL
LIN {X 0,Y 578.649,Z 691.44,A -85,B 0,C 180,E1 1991.8,E2 1991.8} C_VEL
LIN {X 0,Y 571.187,Z 691.44,A -85,B 0,C 180,E1 1995.273,E2 1995.273} C_VEL
LIN {X 0,Y 570.851,Z 691.44,A -85,B 0,C 180,E1 2004.309,E2 2004.309} C_VEL
LIN {X 0,Y 570.397,Z 691.44,A -85,B 0,C 180,E1 2013.06,E2 2013.06} C_VEL
LIN {X 0,Y 570.641,Z 691.44,A -85,B 0,C 180,E1 2020.716,E2 2020.716} C_VEL
LIN {X 0,Y 570.691,Z 691.44,A -85,B 0,C 180,E1 2029.344,E2 2029.344} C_VEL
LIN {X 0,Y 570.716,Z 693.115,A -85,B 0,C 180,E1 2033.822,E2 2033.822} C_VEL
LIN {X 0,Y 577.723,Z 709.297,A -85,B 0,C 180,E1 2034.571,E2 2034.571} C_VEL
LIN {X 0,Y 577.561,Z 784.245,A -85,B 0,C 180,E1 2036.258,E2 2036.258} C_VEL
LIN {X 0,Y 575.83,Z 847.475,A -85,B 0,C 180,E1 2039.234,E2 2039.234} C_VEL
LIN {X 0,Y 573.653,Z 907.821,A -85,B 0,C 180,E1 2043.856,E2 2043.856} C_VEL
LIN {X 0,Y 572.057,Z 955.559,A -85,B 0,C 180,E1 2049.373,E2 2049.373} C_VEL
LIN {X 0,Y 571.305,Z 988.545,A -85,B 0,C 180,E1 2054.989,E2 2054.989} C_VEL
LIN {X 0,Y 571.139,Z 1010.374,A -85,B 0,C 180,E1 2060.826,E2 2060.826} C_VEL
LIN {X 0,Y 571.44,Z 1020.766,A -85,B 0,C 180,E1 2066.192,E2 2066.192} C_VEL
LIN {X 0,Y 571.33,Z 1022.149,A -85,B 0,C 180,E1 2072.283,E2 2072.283} C_VEL
LIN {X 0,Y 571.476,Z 1012.355,A -85,B 0,C 180,E1 2078.398,E2 2078.398} C_VEL
LIN {X 0,Y 571.753,Z 988.551,A -85,B 0,C 180,E1 2084.998,E2 2084.998} C_VEL
LIN {X 0,Y 572.595,Z 949.023,A -85,B 0,C 180,E1 2091.509,E2 2091.509} C_VEL
LIN {X 0,Y 574.23,Z 898.149,A -85,B 0,C 180,E1 2097.015,E2 2097.015} C_VEL
LIN {X 0,Y 576.137,Z 839.326,A -85,B 0,C 180,E1 2101.24,E2 2101.24} C_VEL
LIN {X 0,Y 577.761,Z 775.698,A -85,B 0,C 180,E1 2104.024,E2 2104.024} C_VEL
LIN {X 0,Y 576.106,Z 701.668,A -85,B 0,C 180,E1 2105.658,E2 2105.658} C_VEL
LIN {X 0,Y 571.345,Z 691.44,A -85,B 0,C 180,E1 2106.305,E2 2106.305} C_VEL
LIN {X 0,Y 570.78,Z 691.44,A -85,B 0,C 180,E1 2115.243,E2 2115.243} C_VEL
LIN {X 0,Y 570.625,Z 691.44,A -85,B 0,C 180,E1 2124.208,E2 2124.208} C_VEL
LIN {X 0,Y 570.731,Z 691.44,A -85,B 0,C 180,E1 2132.969,E2 2132.969} C_VEL
LIN {X 0,Y 571.087,Z 691.44,A -85,B 0,C 180,E1 2140.623,E2 2140.623} C_VEL
LIN {X 0,Y 571.005,Z 691.44,A -85,B 0,C 180,E1 2148.523,E2 2148.523} C_VEL
LIN {X 0,Y 570.933,Z 691.44,A -85,B 0,C 180,E1 2156.208,E2 2156.208} C_VEL
LIN {X 0,Y 570.822,Z 691.44,A -85,B 0,C 180,E1 2163.828,E2 2163.828} C_VEL
LIN {X 0,Y 570.721,Z 691.44,A -85,B 0,C 180,E1 2171.519,E2 2171.519} C_VEL
LIN {X 0,Y 570.335,Z 691.44,A -85,B 0,C 180,E1 2177.832,E2 2177.832} C_VEL
LIN {X 0,Y 570.642,Z 693.382,A -85,B 0,C 180,E1 2182.233,E2 2182.233} C_VEL
LIN {X 0,Y 577.752,Z 710.016,A -85,B 0,C 180,E1 2183.012,E2 2183.012} C_VEL
LIN {X 0,Y 576.94,Z 777.538,A -85,B 0,C 180,E1 2185.111,E2 2185.111} C_VEL
LIN {X 0,Y 575.174,Z 839.773,A -85,B 0,C 180,E1 2188.668,E2 2188.668} C_VEL
LIN {X 0,Y 573.329,Z 894.434,A -85,B 0,C 180,E1 2193.51,E2 2193.51} C_VEL
LIN {X 0,Y 572.04,Z 939.656,A -85,B 0,C 180,E1 2199.482,E2 2199.482} C_VEL
LIN {X 0,Y 571.651,Z 971.453,A -85,B 0,C 180,E1 2206.025,E2 2206.025} C_VEL
LIN {X 0,Y 571.232,Z 988.365,A -85,B 0,C 180,E1 2212.41,E2 2212.41} C_VEL
LIN {X 0,Y 571.178,Z 992.827,A -85,B 0,C 180,E1 2218.796,E2 2218.796} C_VEL
LIN {X 0,Y 571.597,Z 983.999,A -85,B 0,C 180,E1 2225.7,E2 2225.7} C_VEL
LIN {X 0,Y 571.783,Z 960.542,A -85,B 0,C 180,E1 2232.513,E2 2232.513} C_VEL
LIN {X 0,Y 572.487,Z 923.334,A -85,B 0,C 180,E1 2238.875,E2 2238.875} C_VEL
LIN {X 0,Y 574.04,Z 873.352,A -85,B 0,C 180,E1 2244.501,E2 2244.501} C_VEL
LIN {X 0,Y 575.988,Z 815.008,A -85,B 0,C 180,E1 2248.868,E2 2248.868} C_VEL
LIN {X 0,Y 577.631,Z 750.745,A -85,B 0,C 180,E1 2251.817,E2 2251.817} C_VEL
LIN {X 0,Y 576.452,Z 703.409,A -85,B 0,C 180,E1 2253.105,E2 2253.105} C_VEL
LIN {X 0,Y 570.948,Z 691.44,A -85,B 0,C 180,E1 2253.811,E2 2253.811} C_VEL
LIN {X 0,Y 570.708,Z 691.44,A -85,B 0,C 180,E1 2261.505,E2 2261.505} C_VEL
LIN {X 0,Y 570.617,Z 691.44,A -85,B 0,C 180,E1 2269.418,E2 2269.418} C_VEL
LIN {X 0,Y 570.548,Z 691.44,A -85,B 0,C 180,E1 2277.742,E2 2277.742} C_VEL
LIN {X 0,Y 570.177,Z 691.44,A -85,B 0,C 180,E1 2285.718,E2 2285.718} C_VEL
LIN {X 0,Y 570.296,Z 691.44,A -85,B 0,C 180,E1 2292.953,E2 2292.953} C_VEL
LIN {X 0,Y 570.643,Z 691.44,A -85,B 0,C 180,E1 2299.329,E2 2299.329} C_VEL
LIN {X 0,Y 570.608,Z 691.44,A -85,B 0,C 180,E1 2308.748,E2 2308.748} C_VEL
LIN {X 0,Y 570.452,Z 691.44,A -85,B 0,C 180,E1 2316.61,E2 2316.61} C_VEL
LIN {X 0,Y 571.603,Z 691.44,A -85,B 0,C 180,E1 2325.715,E2 2325.715} C_VEL
LIN {X 0,Y 571.274,Z 691.44,A -85,B 0,C 180,E1 2335.005,E2 2335.005} C_VEL
LIN {X 0,Y 571.278,Z 691.44,A -85,B 0,C 180,E1 2342.266,E2 2342.266} C_VEL
LIN {X 0,Y 570.972,Z 691.44,A -85,B 0,C 180,E1 2349.928,E2 2349.928} C_VEL
LIN {X 0,Y 571.187,Z 691.44,A -85,B 0,C 180,E1 2355.273,E2 2355.273} C_VEL
LIN {X 0,Y 562.564,Z 691.44,A -85,B 0,C 180,E1 2358.758,E2 2358.758} C_VEL
LIN {X 0,Y 562.369,Z 691.44,A -85,B 0,C 180,E1 2366.413,E2 2366.413} C_VEL
LIN {X 0,Y 562.275,Z 691.44,A -85,B 0,C 180,E1 2373.563,E2 2373.563} C_VEL
LIN {X 0,Y 562.333,Z 691.44,A -85,B 0,C 180,E1 2382.084,E2 2382.084} C_VEL
LIN {X 0,Y 562.318,Z 691.44,A -85,B 0,C 180,E1 2390.637,E2 2390.637} C_VEL
LIN {X 0,Y 562.628,Z 693.45,A -85,B 0,C 180,E1 2393.223,E2 2393.223} C_VEL
LIN {X 0,Y 571.255,Z 712.817,A -85,B 0,C 180,E1 2394.162,E2 2394.162} C_VEL
LIN {X 0,Y 570.815,Z 785.45,A -85,B 0,C 180,E1 2395.846,E2 2395.846} C_VEL
LIN {X 0,Y 568.717,Z 848.595,A -85,B 0,C 180,E1 2398.879,E2 2398.879} C_VEL
LIN {X 0,Y 566.144,Z 908.336,A -85,B 0,C 180,E1 2403.535,E2 2403.535} C_VEL
LIN {X 0,Y 564.321,Z 955.897,A -85,B 0,C 180,E1 2409.125,E2 2409.125} C_VEL
LIN {X 0,Y 563.287,Z 990.326,A -85,B 0,C 180,E1 2415.17,E2 2415.17} C_VEL
LIN {X 0,Y 563.195,Z 1010.374,A -85,B 0,C 180,E1 2420.695,E2 2420.695} C_VEL
LIN {X 0,Y 563.47,Z 1020.766,A -85,B 0,C 180,E1 2426.139,E2 2426.139} C_VEL
LIN {X 0,Y 563.315,Z 1022.15,A -85,B 0,C 180,E1 2432.315,E2 2432.315} C_VEL
LIN {X 0,Y 563.421,Z 1012.356,A -85,B 0,C 180,E1 2438.519,E2 2438.519} C_VEL
LIN {X 0,Y 563.761,Z 988.55,A -85,B 0,C 180,E1 2445.215,E2 2445.215} C_VEL
LIN {X 0,Y 564.804,Z 949.993,A -85,B 0,C 180,E1 2451.685,E2 2451.685} C_VEL
LIN {X 0,Y 566.761,Z 899.301,A -85,B 0,C 180,E1 2457.293,E2 2457.293} C_VEL
LIN {X 0,Y 569.092,Z 840.628,A -85,B 0,C 180,E1 2461.594,E2 2461.594} C_VEL
LIN {X 0,Y 571.101,Z 775.695,A -85,B 0,C 180,E1 2464.477,E2 2464.477} C_VEL
LIN {X 0,Y 569.525,Z 704.792,A -85,B 0,C 180,E1 2466.087,E2 2466.087} C_VEL
LIN {X 0,Y 563.117,Z 691.44,A -85,B 0,C 180,E1 2466.949,E2 2466.949} C_VEL
LIN {X 0,Y 562.466,Z 691.44,A -85,B 0,C 180,E1 2476.565,E2 2476.565} C_VEL
LIN {X 0,Y 562.311,Z 691.44,A -85,B 0,C 180,E1 2485.4,E2 2485.4} C_VEL
LIN {X 0,Y 562.538,Z 691.44,A -85,B 0,C 180,E1 2493.595,E2 2493.595} C_VEL
LIN {X 0,Y 562.758,Z 691.44,A -85,B 0,C 180,E1 2501.957,E2 2501.957} C_VEL
LIN {X 0,Y 562.719,Z 691.44,A -85,B 0,C 180,E1 2509.925,E2 2509.925} C_VEL
LIN {X 0,Y 562.768,Z 691.44,A -85,B 0,C 180,E1 2517.7,E2 2517.7} C_VEL
LIN {X 0,Y 562.83,Z 691.44,A -85,B 0,C 180,E1 2523.882,E2 2523.882} C_VEL
LIN {X 0,Y 562.715,Z 691.44,A -85,B 0,C 180,E1 2531.685,E2 2531.685} C_VEL
LIN {X 0,Y 562.239,Z 691.44,A -85,B 0,C 180,E1 2538.098,E2 2538.098} C_VEL
LIN {X 0,Y 562.428,Z 693.364,A -85,B 0,C 180,E1 2541.629,E2 2541.629} C_VEL
LIN {X 0,Y 571.215,Z 713.179,A -85,B 0,C 180,E1 2542.615,E2 2542.615} C_VEL
LIN {X 0,Y 569.879,Z 782.538,A -85,B 0,C 180,E1 2544.887,E2 2544.887} C_VEL
LIN {X 0,Y 567.764,Z 845.153,A -85,B 0,C 180,E1 2548.662,E2 2548.662} C_VEL
LIN {X 0,Y 565.659,Z 899.301,A -85,B 0,C 180,E1 2553.702,E2 2553.702} C_VEL
LIN {X 0,Y 564.256,Z 943.008,A -85,B 0,C 180,E1 2559.779,E2 2559.779} C_VEL
LIN {X 0,Y 563.844,Z 974.216,A -85,B 0,C 180,E1 2566.66,E2 2566.66} C_VEL
LIN {X 0,Y 563.318,Z 990.184,A -85,B 0,C 180,E1 2573.552,E2 2573.552} C_VEL
LIN {X 0,Y 563.081,Z 992.28,A -85,B 0,C 180,E1 2580.093,E2 2580.093} C_VEL
LIN {X 0,Y 563.168,Z 981.063,A -85,B 0,C 180,E1 2587,E2 2587} C_VEL
LIN {X 0,Y 563.541,Z 956.599,A -85,B 0,C 180,E1 2593.576,E2 2593.576} C_VEL
LIN {X 0,Y 564.664,Z 918.899,A -85,B 0,C 180,E1 2599.798,E2 2599.798} C_VEL
LIN {X 0,Y 566.756,Z 867.79,A -85,B 0,C 180,E1 2605.393,E2 2605.393} C_VEL
LIN {X 0,Y 569.141,Z 808.494,A -85,B 0,C 180,E1 2609.675,E2 2609.675} C_VEL
LIN {X 0,Y 571.143,Z 745.252,A -85,B 0,C 180,E1 2612.446,E2 2612.446} C_VEL
LIN {X 0,Y 569.961,Z 706.404,A -85,B 0,C 180,E1 2613.512,E2 2613.512} C_VEL
LIN {X 0,Y 562.892,Z 691.44,A -85,B 0,C 180,E1 2614.384,E2 2614.384} C_VEL
LIN {X 0,Y 562.703,Z 691.44,A -85,B 0,C 180,E1 2621.671,E2 2621.671} C_VEL
LIN {X 0,Y 562.628,Z 691.44,A -85,B 0,C 180,E1 2629.705,E2 2629.705} C_VEL
LIN {X 0,Y 562.586,Z 691.44,A -85,B 0,C 180,E1 2638.169,E2 2638.169} C_VEL
LIN {X 0,Y 562.509,Z 691.44,A -85,B 0,C 180,E1 2647.376,E2 2647.376} C_VEL
LIN {X 0,Y 562.777,Z 691.44,A -85,B 0,C 180,E1 2656.546,E2 2656.546} C_VEL
LIN {X 0,Y 562.74,Z 691.44,A -85,B 0,C 180,E1 2666.426,E2 2666.426} C_VEL
LIN {X 0,Y 562.831,Z 691.44,A -85,B 0,C 180,E1 2675.283,E2 2675.283} C_VEL
LIN {X 0,Y 563.533,Z 691.44,A -85,B 0,C 180,E1 2685.162,E2 2685.162} C_VEL
LIN {X 0,Y 563.36,Z 691.44,A -85,B 0,C 180,E1 2694.573,E2 2694.573} C_VEL
LIN {X 0,Y 563.27,Z 691.44,A -85,B 0,C 180,E1 2702.298,E2 2702.298} C_VEL
LIN {X 0,Y 562.875,Z 691.44,A -85,B 0,C 180,E1 2710.229,E2 2710.229} C_VEL
LIN {X 0,Y 562.659,Z 691.44,A -85,B 0,C 180,E1 2718.046,E2 2718.046} C_VEL
LIN {X 0,Y 562.564,Z 691.44,A -85,B 0,C 180,E1 2718.758,E2 2718.758} C_VEL
LIN {X 0,Y 554.856,Z 691.44,A -85,B 0,C 180,E1 2722.304,E2 2722.304} C_VEL
LIN {X 0,Y 554.557,Z 691.44,A -85,B 0,C 180,E1 2732.221,E2 2732.221} C_VEL
LIN {X 0,Y 554.461,Z 691.44,A -85,B 0,C 180,E1 2741.175,E2 2741.175} C_VEL
LIN {X 0,Y 554.44,Z 691.44,A -85,B 0,C 180,E1 2749.966,E2 2749.966} C_VEL
LIN {X 0,Y 554.494,Z 693.362,A -85,B 0,C 180,E1 2752.591,E2 2752.591} C_VEL
LIN {X 0,Y 564.778,Z 714.677,A -85,B 0,C 180,E1 2753.715,E2 2753.715} C_VEL
LIN {X 0,Y 564.108,Z 786.091,A -85,B 0,C 180,E1 2755.406,E2 2755.406} C_VEL
LIN {X 0,Y 561.649,Z 849.37,A -85,B 0,C 180,E1 2758.495,E2 2758.495} C_VEL
LIN {X 0,Y 558.764,Z 908.404,A -85,B 0,C 180,E1 2763.164,E2 2763.164} C_VEL
LIN {X 0,Y 556.512,Z 957.345,A -85,B 0,C 180,E1 2769.027,E2 2769.027} C_VEL
LIN {X 0,Y 555.39,Z 990.328,A -85,B 0,C 180,E1 2774.954,E2 2774.954} C_VEL
LIN {X 0,Y 555.265,Z 1010.373,A -85,B 0,C 180,E1 2780.561,E2 2780.561} C_VEL
LIN {X 0,Y 555.477,Z 1020.766,A -85,B 0,C 180,E1 2786.083,E2 2786.083} C_VEL
LIN {X 0,Y 555.301,Z 1022.15,A -85,B 0,C 180,E1 2792.349,E2 2792.349} C_VEL
LIN {X 0,Y 555.368,Z 1012.356,A -85,B 0,C 180,E1 2798.643,E2 2798.643} C_VEL
LIN {X 0,Y 555.765,Z 988.548,A -85,B 0,C 180,E1 2805.44,E2 2805.44} C_VEL
LIN {X 0,Y 557.033,Z 950.508,A -85,B 0,C 180,E1 2811.93,E2 2811.93} C_VEL
LIN {X 0,Y 559.318,Z 899.945,A -85,B 0,C 180,E1 2817.625,E2 2817.625} C_VEL
LIN {X 0,Y 562.073,Z 841.886,A -85,B 0,C 180,E1 2821.959,E2 2821.959} C_VEL
LIN {X 0,Y 564.418,Z 776.801,A -85,B 0,C 180,E1 2824.904,E2 2824.904} C_VEL
LIN {X 0,Y 563.11,Z 707.698,A -85,B 0,C 180,E1 2826.519,E2 2826.519} C_VEL
LIN {X 0,Y 554.879,Z 691.44,A -85,B 0,C 180,E1 2827.623,E2 2827.623} C_VEL
LIN {X 0,Y 554.494,Z 691.44,A -85,B 0,C 180,E1 2836.491,E2 2836.491} C_VEL
LIN {X 0,Y 554.532,Z 691.44,A -85,B 0,C 180,E1 2843.99,E2 2843.99} C_VEL
LIN {X 0,Y 554.569,Z 691.44,A -85,B 0,C 180,E1 2853.186,E2 2853.186} C_VEL
LIN {X 0,Y 554.777,Z 691.44,A -85,B 0,C 180,E1 2861.688,E2 2861.688} C_VEL
LIN {X 0,Y 554.76,Z 691.44,A -85,B 0,C 180,E1 2869.779,E2 2869.779} C_VEL
LIN {X 0,Y 554.768,Z 691.44,A -85,B 0,C 180,E1 2877.667,E2 2877.667} C_VEL
LIN {X 0,Y 554.852,Z 691.44,A -85,B 0,C 180,E1 2883.938,E2 2883.938} C_VEL
LIN {X 0,Y 554.714,Z 691.44,A -85,B 0,C 180,E1 2891.856,E2 2891.856} C_VEL
LIN {X 0,Y 554.04,Z 691.44,A -85,B 0,C 180,E1 2899.093,E2 2899.093} C_VEL
LIN {X 0,Y 554.128,Z 692.263,A -85,B 0,C 180,E1 2900.977,E2 2900.977} C_VEL
LIN {X 0,Y 564.692,Z 716.891,A -85,B 0,C 180,E1 2902.225,E2 2902.225} C_VEL
LIN {X 0,Y 562.977,Z 785.261,A -85,B 0,C 180,E1 2904.559,E2 2904.559} C_VEL
LIN {X 0,Y 560.474,Z 846.599,A -85,B 0,C 180,E1 2908.359,E2 2908.359} C_VEL
LIN {X 0,Y 557.996,Z 900.649,A -85,B 0,C 180,E1 2913.51,E2 2913.51} C_VEL
LIN {X 0,Y 556.382,Z 943.64,A -85,B 0,C 180,E1 2919.623,E2 2919.623} C_VEL
LIN {X 0,Y 555.816,Z 973.762,A -85,B 0,C 180,E1 2926.36,E2 2926.36} C_VEL
LIN {X 0,Y 555.292,Z 989.423,A -85,B 0,C 180,E1 2932.935,E2 2932.935} C_VEL
LIN {X 0,Y 555.019,Z 992.596,A -85,B 0,C 180,E1 2939.613,E2 2939.613} C_VEL
LIN {X 0,Y 555.275,Z 982.227,A -85,B 0,C 180,E1 2946.654,E2 2946.654} C_VEL
LIN {X 0,Y 555.692,Z 958.817,A -85,B 0,C 180,E1 2953.337,E2 2953.337} C_VEL
LIN {X 0,Y 556.875,Z 921.181,A -85,B 0,C 180,E1 2959.798,E2 2959.798} C_VEL
LIN {X 0,Y 559.264,Z 870.577,A -85,B 0,C 180,E1 2965.526,E2 2965.526} C_VEL
LIN {X 0,Y 562.076,Z 811.755,A -85,B 0,C 180,E1 2969.923,E2 2969.923} C_VEL
LIN {X 0,Y 564.432,Z 747.47,A -85,B 0,C 180,E1 2972.838,E2 2972.838} C_VEL
LIN {X 0,Y 563.451,Z 709.533,A -85,B 0,C 180,E1 2973.93,E2 2973.93} C_VEL
LIN {X 0,Y 554.894,Z 691.44,A -85,B 0,C 180,E1 2974.973,E2 2974.973} C_VEL
LIN {X 0,Y 554.703,Z 691.44,A -85,B 0,C 180,E1 2981.841,E2 2981.841} C_VEL
LIN {X 0,Y 554.664,Z 691.44,A -85,B 0,C 180,E1 2990,E2 2990} C_VEL
LIN {X 0,Y 554.67,Z 691.44,A -85,B 0,C 180,E1 2998.608,E2 2998.608} C_VEL
LIN {X 0,Y 554.609,Z 691.44,A -85,B 0,C 180,E1 3008.741,E2 3008.741} C_VEL
LIN {X 0,Y 554.649,Z 691.44,A -85,B 0,C 180,E1 3018.803,E2 3018.803} C_VEL
LIN {X 0,Y 554.636,Z 691.44,A -85,B 0,C 180,E1 3027.741,E2 3027.741} C_VEL
LIN {X 0,Y 554.394,Z 691.44,A -85,B 0,C 180,E1 3036.601,E2 3036.601} C_VEL
LIN {X 0,Y 555.501,Z 691.44,A -85,B 0,C 180,E1 3046.557,E2 3046.557} C_VEL
LIN {X 0,Y 554.97,Z 691.44,A -85,B 0,C 180,E1 3056.063,E2 3056.063} C_VEL
LIN {X 0,Y 554.845,Z 691.44,A -85,B 0,C 180,E1 3063.902,E2 3063.902} C_VEL
LIN {X 0,Y 554.651,Z 691.44,A -85,B 0,C 180,E1 3071.82,E2 3071.82} C_VEL
LIN {X 0,Y 554.603,Z 691.44,A -85,B 0,C 180,E1 3079.977,E2 3079.977} C_VEL
LIN {X 0,Y 554.856,Z 691.44,A -85,B 0,C 180,E1 3082.304,E2 3082.304} C_VEL
LIN {X 0,Y 546.445,Z 691.44,A -85,B 0,C 180,E1 3085.89,E2 3085.89} C_VEL
LIN {X 0,Y 546.411,Z 691.44,A -85,B 0,C 180,E1 3092.761,E2 3092.761} C_VEL
LIN {X 0,Y 546.514,Z 691.44,A -85,B 0,C 180,E1 3100.699,E2 3100.699} C_VEL
LIN {X 0,Y 546.488,Z 691.44,A -85,B 0,C 180,E1 3109.744,E2 3109.744} C_VEL
LIN {X 0,Y 546.461,Z 693.345,A -85,B 0,C 180,E1 3111.944,E2 3111.944} C_VEL
LIN {X 0,Y 558.349,Z 718.612,A -85,B 0,C 180,E1 3113.291,E2 3113.291} C_VEL
LIN {X 0,Y 557.419,Z 788.06,A -85,B 0,C 180,E1 3115.002,E2 3115.002} C_VEL
LIN {X 0,Y 554.509,Z 852.226,A -85,B 0,C 180,E1 3118.235,E2 3118.235} C_VEL
LIN {X 0,Y 551.211,Z 910.439,A -85,B 0,C 180,E1 3122.981,E2 3122.981} C_VEL
LIN {X 0,Y 548.835,Z 957.345,A -85,B 0,C 180,E1 3128.719,E2 3128.719} C_VEL
LIN {X 0,Y 547.415,Z 991.396,A -85,B 0,C 180,E1 3134.979,E2 3134.979} C_VEL
LIN {X 0,Y 546.986,Z 1012.353,A -85,B 0,C 180,E1 3141.222,E2 3141.222} C_VEL
LIN {X 0,Y 546.92,Z 1022.149,A -85,B 0,C 180,E1 3147.614,E2 3147.614} C_VEL
LIN {X 0,Y 547.021,Z 1020.768,A -85,B 0,C 180,E1 3153.976,E2 3153.976} C_VEL
LIN {X 0,Y 546.938,Z 1008.857,A -85,B 0,C 180,E1 3160.115,E2 3160.115} C_VEL
LIN {X 0,Y 547.68,Z 984.621,A -85,B 0,C 180,E1 3166.5,E2 3166.5} C_VEL
LIN {X 0,Y 549.319,Z 947.274,A -85,B 0,C 180,E1 3172.714,E2 3172.714} C_VEL
LIN {X 0,Y 552.09,Z 895.493,A -85,B 0,C 180,E1 3178.449,E2 3178.449} C_VEL
LIN {X 0,Y 555.456,Z 835.235,A -85,B 0,C 180,E1 3182.794,E2 3182.794} C_VEL
LIN {X 0,Y 558.053,Z 771.807,A -85,B 0,C 180,E1 3185.532,E2 3185.532} C_VEL
LIN {X 0,Y 556.712,Z 710.869,A -85,B 0,C 180,E1 3186.958,E2 3186.958} C_VEL
LIN {X 0,Y 546.693,Z 691.44,A -85,B 0,C 180,E1 3188.248,E2 3188.248} C_VEL
LIN {X 0,Y 546.325,Z 691.44,A -85,B 0,C 180,E1 3197.401,E2 3197.401} C_VEL
LIN {X 0,Y 546.265,Z 691.44,A -85,B 0,C 180,E1 3205.316,E2 3205.316} C_VEL
LIN {X 0,Y 546.659,Z 691.44,A -85,B 0,C 180,E1 3212.766,E2 3212.766} C_VEL
LIN {X 0,Y 546.817,Z 691.44,A -85,B 0,C 180,E1 3221.412,E2 3221.412} C_VEL
LIN {X 0,Y 546.722,Z 691.44,A -85,B 0,C 180,E1 3230.196,E2 3230.196} C_VEL
LIN {X 0,Y 546.786,Z 691.44,A -85,B 0,C 180,E1 3237.633,E2 3237.633} C_VEL
LIN {X 0,Y 546.846,Z 691.44,A -85,B 0,C 180,E1 3243.996,E2 3243.996} C_VEL
LIN {X 0,Y 546.715,Z 691.44,A -85,B 0,C 180,E1 3252.032,E2 3252.032} C_VEL
LIN {X 0,Y 545.996,Z 691.44,A -85,B 0,C 180,E1 3260.225,E2 3260.225} C_VEL
LIN {X 0,Y 558.132,Z 719.852,A -85,B 0,C 180,E1 3261.811,E2 3261.811} C_VEL
LIN {X 0,Y 556.037,Z 788.169,A -85,B 0,C 180,E1 3264.239,E2 3264.239} C_VEL
LIN {X 0,Y 553.126,Z 849.924,A -85,B 0,C 180,E1 3268.198,E2 3268.198} C_VEL
LIN {X 0,Y 550.349,Z 901.986,A -85,B 0,C 180,E1 3273.312,E2 3273.312} C_VEL
LIN {X 0,Y 548.52,Z 945.107,A -85,B 0,C 180,E1 3279.617,E2 3279.617} C_VEL
LIN {X 0,Y 547.843,Z 974.624,A -85,B 0,C 180,E1 3286.446,E2 3286.446} C_VEL
LIN {X 0,Y 547.299,Z 990.16,A -85,B 0,C 180,E1 3293.405,E2 3293.405} C_VEL
LIN {X 0,Y 546.967,Z 992.771,A -85,B 0,C 180,E1 3299.117,E2 3299.117} C_VEL
LIN {X 0,Y 547.411,Z 983.389,A -85,B 0,C 180,E1 3306.298,E2 3306.298} C_VEL
LIN {X 0,Y 547.813,Z 960.87,A -85,B 0,C 180,E1 3313.09,E2 3313.09} C_VEL
LIN {X 0,Y 549.043,Z 924.472,A -85,B 0,C 180,E1 3319.651,E2 3319.651} C_VEL
LIN {X 0,Y 551.742,Z 874.395,A -85,B 0,C 180,E1 3325.564,E2 3325.564} C_VEL
LIN {X 0,Y 554.932,Z 815.446,A -85,B 0,C 180,E1 3330.151,E2 3330.151} C_VEL
LIN {X 0,Y 557.659,Z 751.503,A -85,B 0,C 180,E1 3333.18,E2 3333.18} C_VEL
LIN {X 0,Y 556.922,Z 712.421,A -85,B 0,C 180,E1 3334.36,E2 3334.36} C_VEL
LIN {X 0,Y 546.947,Z 691.44,A -85,B 0,C 180,E1 3335.574,E2 3335.574} C_VEL
LIN {X 0,Y 546.932,Z 691.44,A -85,B 0,C 180,E1 3343.643,E2 3343.643} C_VEL
LIN {X 0,Y 546.932,Z 691.44,A -85,B 0,C 180,E1 3353.725,E2 3353.725} C_VEL
LIN {X 0,Y 546.474,Z 691.44,A -85,B 0,C 180,E1 3362.789,E2 3362.789} C_VEL
LIN {X 0,Y 546.56,Z 691.44,A -85,B 0,C 180,E1 3370.732,E2 3370.732} C_VEL
LIN {X 0,Y 546.407,Z 691.44,A -85,B 0,C 180,E1 3379.8,E2 3379.8} C_VEL
LIN {X 0,Y 546.418,Z 691.44,A -85,B 0,C 180,E1 3389.069,E2 3389.069} C_VEL
LIN {X 0,Y 546.498,Z 691.44,A -85,B 0,C 180,E1 3396.242,E2 3396.242} C_VEL
LIN {X 0,Y 547.513,Z 691.44,A -85,B 0,C 180,E1 3406.357,E2 3406.357} C_VEL
LIN {X 0,Y 546.977,Z 691.44,A -85,B 0,C 180,E1 3416.005,E2 3416.005} C_VEL
LIN {X 0,Y 546.836,Z 691.44,A -85,B 0,C 180,E1 3423.959,E2 3423.959} C_VEL
LIN {X 0,Y 546.654,Z 691.44,A -85,B 0,C 180,E1 3431.996,E2 3431.996} C_VEL
LIN {X 0,Y 546.621,Z 691.44,A -85,B 0,C 180,E1 3440.281,E2 3440.281} C_VEL
LIN {X 0,Y 546.445,Z 691.44,A -85,B 0,C 180,E1 3445.89,E2 3445.89} C_VEL
LIN {X 0,Y 538.564,Z 691.44,A -85,B 0,C 180,E1 3449.542,E2 3449.542} C_VEL
LIN {X 0,Y 538.513,Z 691.44,A -85,B 0,C 180,E1 3459.316,E2 3459.316} C_VEL
LIN {X 0,Y 538.564,Z 691.44,A -85,B 0,C 180,E1 3468.532,E2 3468.532} C_VEL
LIN {X 0,Y 538.406,Z 692.913,A -85,B 0,C 180,E1 3471.262,E2 3471.262} C_VEL
LIN {X 0,Y 551.991,Z 721.977,A -85,B 0,C 180,E1 3472.851,E2 3472.851} C_VEL
LIN {X 0,Y 550.71,Z 790.707,A -85,B 0,C 180,E1 3474.624,E2 3474.624} C_VEL
LIN {X 0,Y 547.447,Z 853.618,A -85,B 0,C 180,E1 3477.873,E2 3477.873} C_VEL
LIN {X 0,Y 543.738,Z 911.642,A -85,B 0,C 180,E1 3482.707,E2 3482.707} C_VEL
LIN {X 0,Y 541.024,Z 958.697,A -85,B 0,C 180,E1 3488.613,E2 3488.613} C_VEL
LIN {X 0,Y 539.469,Z 992.093,A -85,B 0,C 180,E1 3494.917,E2 3494.917} C_VEL
LIN {X 0,Y 539.035,Z 1012.353,A -85,B 0,C 180,E1 3501.091,E2 3501.091} C_VEL
LIN {X 0,Y 538.941,Z 1022.149,A -85,B 0,C 180,E1 3507.578,E2 3507.578} C_VEL
LIN {X 0,Y 539.039,Z 1020.768,A -85,B 0,C 180,E1 3514.035,E2 3514.035} C_VEL
LIN {X 0,Y 538.952,Z 1009.3,A -85,B 0,C 180,E1 3520.109,E2 3520.109} C_VEL
LIN {X 0,Y 539.769,Z 986.592,A -85,B 0,C 180,E1 3526.328,E2 3526.328} C_VEL
LIN {X 0,Y 541.575,Z 950.057,A -85,B 0,C 180,E1 3532.657,E2 3532.657} C_VEL
LIN {X 0,Y 544.57,Z 899.226,A -85,B 0,C 180,E1 3538.511,E2 3538.511} C_VEL
LIN {X 0,Y 548.259,Z 841.05,A -85,B 0,C 180,E1 3542.917,E2 3542.917} C_VEL
LIN {X 0,Y 551.292,Z 776.869,A -85,B 0,C 180,E1 3545.859,E2 3545.859} C_VEL
LIN {X 0,Y 550.524,Z 714.354,A -85,B 0,C 180,E1 3547.388,E2 3547.388} C_VEL
LIN {X 0,Y 538.533,Z 691.44,A -85,B 0,C 180,E1 3548.835,E2 3548.835} C_VEL
LIN {X 0,Y 538.386,Z 691.44,A -85,B 0,C 180,E1 3556.362,E2 3556.362} C_VEL
LIN {X 0,Y 538.338,Z 691.44,A -85,B 0,C 180,E1 3564.73,E2 3564.73} C_VEL
LIN {X 0,Y 538.362,Z 691.44,A -85,B 0,C 180,E1 3574.119,E2 3574.119} C_VEL
LIN {X 0,Y 538.614,Z 691.44,A -85,B 0,C 180,E1 3582.816,E2 3582.816} C_VEL
LIN {X 0,Y 538.755,Z 691.44,A -85,B 0,C 180,E1 3591.109,E2 3591.109} C_VEL
LIN {X 0,Y 539.019,Z 691.44,A -85,B 0,C 180,E1 3599.212,E2 3599.212} C_VEL
LIN {X 0,Y 539.309,Z 691.44,A -85,B 0,C 180,E1 3608.92,E2 3608.92} C_VEL
LIN {X 0,Y 538.564,Z 691.44,A -85,B 0,C 180,E1 3617.225,E2 3617.225} C_VEL
LIN {X 0,Y 538.081,Z 692.52,A -85,B 0,C 180,E1 3619.684,E2 3619.684} C_VEL
LIN {X 0,Y 551.609,Z 723.185,A -85,B 0,C 180,E1 3621.397,E2 3621.397} C_VEL
LIN {X 0,Y 549.13,Z 791.025,A -85,B 0,C 180,E1 3623.911,E2 3623.911} C_VEL
LIN {X 0,Y 545.763,Z 852.888,A -85,B 0,C 180,E1 3628.006,E2 3628.006} C_VEL
LIN {X 0,Y 542.605,Z 906.473,A -85,B 0,C 180,E1 3633.498,E2 3633.498} C_VEL
LIN {X 0,Y 540.662,Z 948.76,A -85,B 0,C 180,E1 3640.042,E2 3640.042} C_VEL
LIN {X 0,Y 539.788,Z 976.757,A -85,B 0,C 180,E1 3646.954,E2 3646.954} C_VEL
LIN {X 0,Y 539.305,Z 990.151,A -85,B 0,C 180,E1 3653.332,E2 3653.332} C_VEL
LIN {X 0,Y 538.843,Z 992.109,A -85,B 0,C 180,E1 3660.472,E2 3660.472} C_VEL
LIN {X 0,Y 539.253,Z 982.28,A -85,B 0,C 180,E1 3666.893,E2 3666.893} C_VEL
LIN {X 0,Y 539.77,Z 959.376,A -85,B 0,C 180,E1 3673.672,E2 3673.672} C_VEL
LIN {X 0,Y 541.372,Z 922.133,A -85,B 0,C 180,E1 3680.318,E2 3680.318} C_VEL
LIN {X 0,Y 544.496,Z 871.957,A -85,B 0,C 180,E1 3686.205,E2 3686.205} C_VEL
LIN {X 0,Y 548.134,Z 812.421,A -85,B 0,C 180,E1 3690.794,E2 3690.794} C_VEL
LIN {X 0,Y 551.214,Z 748.87,A -85,B 0,C 180,E1 3693.751,E2 3693.751} C_VEL
LIN {X 0,Y 550.413,Z 715.441,A -85,B 0,C 180,E1 3694.796,E2 3694.796} C_VEL
LIN {X 0,Y 539.029,Z 691.44,A -85,B 0,C 180,E1 3696.325,E2 3696.325} C_VEL
LIN {X 0,Y 539.122,Z 691.44,A -85,B 0,C 180,E1 3705.511,E2 3705.511} C_VEL
LIN {X 0,Y 538.841,Z 691.44,A -85,B 0,C 180,E1 3714.104,E2 3714.104} C_VEL
LIN {X 0,Y 538.313,Z 691.44,A -85,B 0,C 180,E1 3723.35,E2 3723.35} C_VEL
LIN {X 0,Y 538.371,Z 691.44,A -85,B 0,C 180,E1 3731.657,E2 3731.657} C_VEL
LIN {X 0,Y 538.188,Z 691.44,A -85,B 0,C 180,E1 3740.608,E2 3740.608} C_VEL
LIN {X 0,Y 538.386,Z 691.44,A -85,B 0,C 180,E1 3749.288,E2 3749.288} C_VEL
LIN {X 0,Y 538.119,Z 691.44,A -85,B 0,C 180,E1 3757.607,E2 3757.607} C_VEL
LIN {X 0,Y 539.498,Z 691.44,A -85,B 0,C 180,E1 3766.151,E2 3766.151} C_VEL
LIN {X 0,Y 538.983,Z 691.44,A -85,B 0,C 180,E1 3775.946,E2 3775.946} C_VEL
LIN {X 0,Y 538.845,Z 691.44,A -85,B 0,C 180,E1 3784.018,E2 3784.018} C_VEL
LIN {X 0,Y 538.662,Z 691.44,A -85,B 0,C 180,E1 3792.176,E2 3792.176} C_VEL
LIN {X 0,Y 538.656,Z 691.44,A -85,B 0,C 180,E1 3800.595,E2 3800.595} C_VEL
LIN {X 0,Y 538.564,Z 691.44,A -85,B 0,C 180,E1 3809.542,E2 3809.542} C_VEL
LIN {X 0,Y 530.215,Z 691.44,A -85,B 0,C 180,E1 3813.259,E2 3813.259} C_VEL
LIN {X 0,Y 530.247,Z 691.44,A -85,B 0,C 180,E1 3822.228,E2 3822.228} C_VEL
LIN {X 0,Y 530.489,Z 693.076,A -85,B 0,C 180,E1 3830.576,E2 3830.576} C_VEL
LIN {X 0,Y 545.641,Z 724.641,A -85,B 0,C 180,E1 3832.387,E2 3832.387} C_VEL
LIN {X 0,Y 544.057,Z 792.131,A -85,B 0,C 180,E1 3834.188,E2 3834.188} C_VEL
LIN {X 0,Y 540.367,Z 855.929,A -85,B 0,C 180,E1 3837.563,E2 3837.563} C_VEL
LIN {X 0,Y 536.163,Z 914.293,A -85,B 0,C 180,E1 3842.577,E2 3842.577} C_VEL
LIN {X 0,Y 533.194,Z 960.044,A -85,B 0,C 180,E1 3848.502,E2 3848.502} C_VEL
LIN {X 0,Y 531.601,Z 992.092,A -85,B 0,C 180,E1 3854.688,E2 3854.688} C_VEL
LIN {X 0,Y 531.087,Z 1012.353,A -85,B 0,C 180,E1 3860.957,E2 3860.957} C_VEL
LIN {X 0,Y 530.977,Z 1022.149,A -85,B 0,C 180,E1 3867.542,E2 3867.542} C_VEL
LIN {X 0,Y 531.027,Z 1020.768,A -85,B 0,C 180,E1 3874.096,E2 3874.096} C_VEL
LIN {X 0,Y 530.981,Z 1009.517,A -85,B 0,C 180,E1 3880.184,E2 3880.184} C_VEL
LIN {X 0,Y 531.854,Z 985.487,A -85,B 0,C 180,E1 3886.819,E2 3886.819} C_VEL
LIN {X 0,Y 533.927,Z 948.549,A -85,B 0,C 180,E1 3893.226,E2 3893.226} C_VEL
LIN {X 0,Y 537.456,Z 897.168,A -85,B 0,C 180,E1 3899.13,E2 3899.13} C_VEL
LIN {X 0,Y 541.547,Z 838.332,A -85,B 0,C 180,E1 3903.551,E2 3903.551} C_VEL
LIN {X 0,Y 544.909,Z 774.415,A -85,B 0,C 180,E1 3906.438,E2 3906.438} C_VEL
LIN {X 0,Y 544.301,Z 717.522,A -85,B 0,C 180,E1 3907.838,E2 3907.838} C_VEL
LIN {X 0,Y 530.411,Z 691.44,A -85,B 0,C 180,E1 3909.681,E2 3909.681} C_VEL
LIN {X 0,Y 530.231,Z 691.44,A -85,B 0,C 180,E1 3917.77,E2 3917.77} C_VEL
LIN {X 0,Y 530.195,Z 691.44,A -85,B 0,C 180,E1 3926.104,E2 3926.104} C_VEL
LIN {X 0,Y 530.348,Z 691.44,A -85,B 0,C 180,E1 3934.338,E2 3934.338} C_VEL
LIN {X 0,Y 530.606,Z 691.44,A -85,B 0,C 180,E1 3943.36,E2 3943.36} C_VEL
LIN {X 0,Y 531.065,Z 691.44,A -85,B 0,C 180,E1 3952.633,E2 3952.633} C_VEL
LIN {X 0,Y 531.208,Z 691.44,A -85,B 0,C 180,E1 3962.474,E2 3962.474} C_VEL
LIN {X 0,Y 530.875,Z 691.44,A -85,B 0,C 180,E1 3970.725,E2 3970.725} C_VEL
LIN {X 0,Y 530.207,Z 692.897,A -85,B 0,C 180,E1 3979.016,E2 3979.016} C_VEL
LIN {X 0,Y 545.145,Z 726.238,A -85,B 0,C 180,E1 3980.97,E2 3980.97} C_VEL
LIN {X 0,Y 542.213,Z 794.233,A -85,B 0,C 180,E1 3983.595,E2 3983.595} C_VEL
LIN {X 0,Y 538.453,Z 854.765,A -85,B 0,C 180,E1 3987.727,E2 3987.727} C_VEL
LIN {X 0,Y 534.937,Z 908.133,A -85,B 0,C 180,E1 3993.337,E2 3993.337} C_VEL
LIN {X 0,Y 532.776,Z 949.29,A -85,B 0,C 180,E1 3999.872,E2 3999.872} C_VEL
LIN {X 0,Y 531.731,Z 977.671,A -85,B 0,C 180,E1 4007.113,E2 4007.113} C_VEL
LIN {X 0,Y 531.075,Z 991.48,A -85,B 0,C 180,E1 4014.542,E2 4014.542} C_VEL
LIN {X 0,Y 530.803,Z 991.003,A -85,B 0,C 180,E1 4021.853,E2 4021.853} C_VEL
LIN {X 0,Y 530.965,Z 979.147,A -85,B 0,C 180,E1 4028.281,E2 4028.281} C_VEL
LIN {X 0,Y 531.784,Z 957.824,A -85,B 0,C 180,E1 4034.271,E2 4034.271} C_VEL
LIN {X 0,Y 533.69,Z 921.207,A -85,B 0,C 180,E1 4040.797,E2 4040.797} C_VEL
LIN {X 0,Y 537.216,Z 870.585,A -85,B 0,C 180,E1 4046.762,E2 4046.762} C_VEL
LIN {X 0,Y 541.304,Z 811.742,A -85,B 0,C 180,E1 4051.306,E2 4051.306} C_VEL
LIN {X 0,Y 544.687,Z 749.31,A -85,B 0,C 180,E1 4054.232,E2 4054.232} C_VEL
LIN {X 0,Y 544.016,Z 718.736,A -85,B 0,C 180,E1 4055.222,E2 4055.222} C_VEL
LIN {X 0,Y 531.127,Z 691.44,A -85,B 0,C 180,E1 4056.976,E2 4056.976} C_VEL
LIN {X 0,Y 530.851,Z 691.44,A -85,B 0,C 180,E1 4067.469,E2 4067.469} C_VEL
LIN {X 0,Y 530.534,Z 691.44,A -85,B 0,C 180,E1 4076.32,E2 4076.32} C_VEL
LIN {X 0,Y 530.184,Z 691.44,A -85,B 0,C 180,E1 4085.323,E2 4085.323} C_VEL
LIN {X 0,Y 530.294,Z 691.44,A -85,B 0,C 180,E1 4094.52,E2 4094.52} C_VEL
LIN {X 0,Y 530.213,Z 691.44,A -85,B 0,C 180,E1 4104.06,E2 4104.06} C_VEL
LIN {X 0,Y 530.67,Z 691.44,A -85,B 0,C 180,E1 4113.674,E2 4113.674} C_VEL
LIN {X 0,Y 531.232,Z 691.44,A -85,B 0,C 180,E1 4124.237,E2 4124.237} C_VEL
LIN {X 0,Y 531.276,Z 691.44,A -85,B 0,C 180,E1 4134.245,E2 4134.245} C_VEL
LIN {X 0,Y 531.207,Z 691.44,A -85,B 0,C 180,E1 4142.436,E2 4142.436} C_VEL
LIN {X 0,Y 530.809,Z 691.44,A -85,B 0,C 180,E1 4150.688,E2 4150.688} C_VEL
LIN {X 0,Y 530.57,Z 691.44,A -85,B 0,C 180,E1 4159.179,E2 4159.179} C_VEL
LIN {X 0,Y 530.395,Z 691.44,A -85,B 0,C 180,E1 4168.142,E2 4168.142} C_VEL
LIN {X 0,Y 530.215,Z 691.44,A -85,B 0,C 180,E1 4173.259,E2 4173.259} C_VEL
LIN {X 0,Y 522.149,Z 691.44,A -85,B 0,C 180,E1 4177.004,E2 4177.004} C_VEL
LIN {X 0,Y 522.472,Z 691.44,A -85,B 0,C 180,E1 4186.953,E2 4186.953} C_VEL
LIN {X 0,Y 522.46,Z 692.88,A -85,B 0,C 180,E1 4189.845,E2 4189.845} C_VEL
LIN {X 0,Y 539.357,Z 728.739,A -85,B 0,C 180,E1 4191.939,E2 4191.939} C_VEL
LIN {X 0,Y 537.32,Z 795.689,A -85,B 0,C 180,E1 4193.827,E2 4193.827} C_VEL
LIN {X 0,Y 533.304,Z 858.035,A -85,B 0,C 180,E1 4197.233,E2 4197.233} C_VEL
LIN {X 0,Y 528.585,Z 916.861,A -85,B 0,C 180,E1 4202.434,E2 4202.434} C_VEL
LIN {X 0,Y 525.211,Z 962.822,A -85,B 0,C 180,E1 4208.621,E2 4208.621} C_VEL
LIN {X 0,Y 523.562,Z 993.836,A -85,B 0,C 180,E1 4214.877,E2 4214.877} C_VEL
LIN {X 0,Y 522.947,Z 1014.285,A -85,B 0,C 180,E1 4221.656,E2 4221.656} C_VEL
LIN {X 0,Y 522.986,Z 1022.149,A -85,B 0,C 180,E1 4227.505,E2 4227.505} C_VEL
LIN {X 0,Y 523.05,Z 1020.769,A -85,B 0,C 180,E1 4234.159,E2 4234.159} C_VEL
LIN {X 0,Y 522.969,Z 1009.3,A -85,B 0,C 180,E1 4240.421,E2 4240.421} C_VEL
LIN {X 0,Y 523.929,Z 985.921,A -85,B 0,C 180,E1 4246.985,E2 4246.985} C_VEL
LIN {X 0,Y 526.179,Z 950.027,A -85,B 0,C 180,E1 4253.363,E2 4253.363} C_VEL
LIN {X 0,Y 530.012,Z 899.404,A -85,B 0,C 180,E1 4259.351,E2 4259.351} C_VEL
LIN {X 0,Y 534.585,Z 840.741,A -85,B 0,C 180,E1 4263.891,E2 4263.891} C_VEL
LIN {X 0,Y 538.303,Z 776.906,A -85,B 0,C 180,E1 4266.863,E2 4266.863} C_VEL
LIN {X 0,Y 537.939,Z 720.643,A -85,B 0,C 180,E1 4268.314,E2 4268.314} C_VEL
LIN {X 0,Y 522.38,Z 691.44,A -85,B 0,C 180,E1 4270.295,E2 4270.295} C_VEL
LIN {X 0,Y 522.233,Z 691.44,A -85,B 0,C 180,E1 4279.206,E2 4279.206} C_VEL
LIN {X 0,Y 522.301,Z 691.44,A -85,B 0,C 180,E1 4288.996,E2 4288.996} C_VEL
LIN {X 0,Y 522.735,Z 691.44,A -85,B 0,C 180,E1 4298.748,E2 4298.748} C_VEL
LIN {X 0,Y 522.999,Z 691.44,A -85,B 0,C 180,E1 4307.453,E2 4307.453} C_VEL
LIN {X 0,Y 523.026,Z 691.44,A -85,B 0,C 180,E1 4315.86,E2 4315.86} C_VEL
LIN {X 0,Y 522.85,Z 691.44,A -85,B 0,C 180,E1 4324.179,E2 4324.179} C_VEL
LIN {X 0,Y 522.745,Z 691.44,A -85,B 0,C 180,E1 4332.593,E2 4332.593} C_VEL
LIN {X 0,Y 522.474,Z 693.439,A -85,B 0,C 180,E1 4338.337,E2 4338.337} C_VEL
LIN {X 0,Y 538.685,Z 728.854,A -85,B 0,C 180,E1 4340.526,E2 4340.526} C_VEL
LIN {X 0,Y 535.314,Z 796.838,A -85,B 0,C 180,E1 4343.24,E2 4343.24} C_VEL
LIN {X 0,Y 531.091,Z 857.567,A -85,B 0,C 180,E1 4347.521,E2 4347.521} C_VEL
LIN {X 0,Y 527.308,Z 908.995,A -85,B 0,C 180,E1 4353.076,E2 4353.076} C_VEL
LIN {X 0,Y 524.863,Z 950.116,A -85,B 0,C 180,E1 4359.757,E2 4359.757} C_VEL
LIN {X 0,Y 523.76,Z 978.057,A -85,B 0,C 180,E1 4367.086,E2 4367.086} C_VEL
LIN {X 0,Y 523.264,Z 990.514,A -85,B 0,C 180,E1 4373.52,E2 4373.52} C_VEL
LIN {X 0,Y 522.801,Z 992.712,A -85,B 0,C 180,E1 4379.471,E2 4379.471} C_VEL
LIN {X 0,Y 523.359,Z 983.909,A -85,B 0,C 180,E1 4386.46,E2 4386.46} C_VEL
LIN {X 0,Y 523.906,Z 961.237,A -85,B 0,C 180,E1 4393.711,E2 4393.711} C_VEL
LIN {X 0,Y 525.801,Z 925.866,A -85,B 0,C 180,E1 4400.448,E2 4400.448} C_VEL
LIN {X 0,Y 529.564,Z 876.41,A -85,B 0,C 180,E1 4406.612,E2 4406.612} C_VEL
LIN {X 0,Y 534.092,Z 817.555,A -85,B 0,C 180,E1 4411.425,E2 4411.425} C_VEL
LIN {X 0,Y 537.981,Z 753.346,A -85,B 0,C 180,E1 4414.604,E2 4414.604} C_VEL
LIN {X 0,Y 537.397,Z 721.151,A -85,B 0,C 180,E1 4415.699,E2 4415.699} C_VEL
LIN {X 0,Y 523.173,Z 691.44,A -85,B 0,C 180,E1 4417.711,E2 4417.711} C_VEL
LIN {X 0,Y 522.781,Z 691.44,A -85,B 0,C 180,E1 4427.747,E2 4427.747} C_VEL
LIN {X 0,Y 522.474,Z 691.44,A -85,B 0,C 180,E1 4436.758,E2 4436.758} C_VEL
LIN {X 0,Y 522.196,Z 691.44,A -85,B 0,C 180,E1 4444.522,E2 4444.522} C_VEL
LIN {X 0,Y 522.242,Z 691.44,A -85,B 0,C 180,E1 4453.071,E2 4453.071} C_VEL
LIN {X 0,Y 522.051,Z 691.44,A -85,B 0,C 180,E1 4461.304,E2 4461.304} C_VEL
LIN {X 0,Y 522.312,Z 691.44,A -85,B 0,C 180,E1 4469.424,E2 4469.424} C_VEL
LIN {X 0,Y 522.217,Z 691.44,A -85,B 0,C 180,E1 4476.886,E2 4476.886} C_VEL
LIN {X 0,Y 523.379,Z 691.44,A -85,B 0,C 180,E1 4486.259,E2 4486.259} C_VEL
LIN {X 0,Y 523.015,Z 691.44,A -85,B 0,C 180,E1 4495.822,E2 4495.822} C_VEL
LIN {X 0,Y 523.216,Z 691.44,A -85,B 0,C 180,E1 4502.474,E2 4502.474} C_VEL
LIN {X 0,Y 522.776,Z 691.44,A -85,B 0,C 180,E1 4510.854,E2 4510.854} C_VEL
LIN {X 0,Y 522.55,Z 691.44,A -85,B 0,C 180,E1 4519.485,E2 4519.485} C_VEL
LIN {X 0,Y 522.419,Z 691.44,A -85,B 0,C 180,E1 4528.611,E2 4528.611} C_VEL
LIN {X 0,Y 522.149,Z 691.44,A -85,B 0,C 180,E1 4537.004,E2 4537.004} C_VEL
LIN {X 0,Y 514.245,Z 691.44,A -85,B 0,C 180,E1 4540.845,E2 4540.845} C_VEL
LIN {X 0,Y 514.626,Z 693.142,A -85,B 0,C 180,E1 4549.129,E2 4549.129} C_VEL
LIN {X 0,Y 533.073,Z 730.096,A -85,B 0,C 180,E1 4551.434,E2 4551.434} C_VEL
LIN {X 0,Y 530.749,Z 796.801,A -85,B 0,C 180,E1 4553.357,E2 4553.357} C_VEL
LIN {X 0,Y 526.361,Z 858.033,A -85,B 0,C 180,E1 4556.746,E2 4556.746} C_VEL
LIN {X 0,Y 521.349,Z 915.732,A -85,B 0,C 180,E1 4561.891,E2 4561.891} C_VEL
LIN {X 0,Y 517.617,Z 962.078,A -85,B 0,C 180,E1 4568.165,E2 4568.165} C_VEL
LIN {X 0,Y 515.709,Z 993.835,A -85,B 0,C 180,E1 4574.641,E2 4574.641} C_VEL
LIN {X 0,Y 515.005,Z 1014.285,A -85,B 0,C 180,E1 4581.527,E2 4581.527} C_VEL
LIN {X 0,Y 514.993,Z 1022.15,A -85,B 0,C 180,E1 4587.466,E2 4587.466} C_VEL
LIN {X 0,Y 515.042,Z 1020.769,A -85,B 0,C 180,E1 4594.224,E2 4594.224} C_VEL
LIN {X 0,Y 514.976,Z 1009.216,A -85,B 0,C 180,E1 4600.616,E2 4600.616} C_VEL
LIN {X 0,Y 516.021,Z 986.116,A -85,B 0,C 180,E1 4607.209,E2 4607.209} C_VEL
LIN {X 0,Y 518.537,Z 950.029,A -85,B 0,C 180,E1 4613.729,E2 4613.729} C_VEL
LIN {X 0,Y 522.761,Z 899.989,A -85,B 0,C 180,E1 4619.738,E2 4619.738} C_VEL
LIN {X 0,Y 527.71,Z 841.878,A -85,B 0,C 180,E1 4624.319,E2 4624.319} C_VEL
LIN {X 0,Y 531.736,Z 778.828,A -85,B 0,C 180,E1 4627.321,E2 4627.321} C_VEL
LIN {X 0,Y 531.757,Z 723.902,A -85,B 0,C 180,E1 4628.787,E2 4628.787} C_VEL
LIN {X 0,Y 514.374,Z 691.44,A -85,B 0,C 180,E1 4631.019,E2 4631.019} C_VEL
LIN {X 0,Y 514.291,Z 691.44,A -85,B 0,C 180,E1 4640.659,E2 4640.659} C_VEL
LIN {X 0,Y 514.454,Z 691.44,A -85,B 0,C 180,E1 4650.904,E2 4650.904} C_VEL
LIN {X 0,Y 514.769,Z 691.44,A -85,B 0,C 180,E1 4660.208,E2 4660.208} C_VEL
LIN {X 0,Y 514.815,Z 691.44,A -85,B 0,C 180,E1 4668.976,E2 4668.976} C_VEL
LIN {X 0,Y 514.81,Z 691.44,A -85,B 0,C 180,E1 4677.486,E2 4677.486} C_VEL
LIN {X 0,Y 514.846,Z 691.44,A -85,B 0,C 180,E1 4684.245,E2 4684.245} C_VEL
LIN {X 0,Y 514.767,Z 691.44,A -85,B 0,C 180,E1 4692.791,E2 4692.791} C_VEL
LIN {X 0,Y 514.601,Z 693.22,A -85,B 0,C 180,E1 4697.614,E2 4697.614} C_VEL
LIN {X 0,Y 532.222,Z 732.036,A -85,B 0,C 180,E1 4700.089,E2 4700.089} C_VEL
LIN {X 0,Y 528.43,Z 799.549,A -85,B 0,C 180,E1 4702.89,E2 4702.89} C_VEL
LIN {X 0,Y 523.726,Z 860.504,A -85,B 0,C 180,E1 4707.325,E2 4707.325} C_VEL
LIN {X 0,Y 519.521,Z 912.401,A -85,B 0,C 180,E1 4713.16,E2 4713.16} C_VEL
LIN {X 0,Y 516.947,Z 952.164,A -85,B 0,C 180,E1 4719.893,E2 4719.893} C_VEL
LIN {X 0,Y 515.622,Z 979.232,A -85,B 0,C 180,E1 4727.35,E2 4727.35} C_VEL
LIN {X 0,Y 514.949,Z 991.877,A -85,B 0,C 180,E1 4734.924,E2 4734.924} C_VEL
LIN {X 0,Y 514.734,Z 991.933,A -85,B 0,C 180,E1 4740.892,E2 4740.892} C_VEL
LIN {X 0,Y 515.143,Z 982.044,A -85,B 0,C 180,E1 4747.421,E2 4747.421} C_VEL
LIN {X 0,Y 515.94,Z 960.21,A -85,B 0,C 180,E1 4754.213,E2 4754.213} C_VEL
LIN {X 0,Y 518.134,Z 924.966,A -85,B 0,C 180,E1 4760.943,E2 4760.943} C_VEL
LIN {X 0,Y 522.35,Z 875.056,A -85,B 0,C 180,E1 4767.191,E2 4767.191} C_VEL
LIN {X 0,Y 527.308,Z 816.923,A -85,B 0,C 180,E1 4771.959,E2 4771.959} C_VEL
LIN {X 0,Y 531.545,Z 753.421,A -85,B 0,C 180,E1 4775.12,E2 4775.12} C_VEL
LIN {X 0,Y 531.157,Z 724.648,A -85,B 0,C 180,E1 4776.129,E2 4776.129} C_VEL
LIN {X 0,Y 515.18,Z 691.44,A -85,B 0,C 180,E1 4778.445,E2 4778.445} C_VEL
LIN {X 0,Y 514.725,Z 691.44,A -85,B 0,C 180,E1 4788.035,E2 4788.035} C_VEL
LIN {X 0,Y 514.475,Z 691.44,A -85,B 0,C 180,E1 4797.209,E2 4797.209} C_VEL
LIN {X 0,Y 514.122,Z 691.44,A -85,B 0,C 180,E1 4805.719,E2 4805.719} C_VEL
LIN {X 0,Y 514.24,Z 691.44,A -85,B 0,C 180,E1 4813.91,E2 4813.91} C_VEL
LIN {X 0,Y 514.047,Z 691.44,A -85,B 0,C 180,E1 4822.742,E2 4822.742} C_VEL
LIN {X 0,Y 514.289,Z 691.44,A -85,B 0,C 180,E1 4830.849,E2 4830.849} C_VEL
LIN {X 0,Y 514.084,Z 691.44,A -85,B 0,C 180,E1 4840.139,E2 4840.139} C_VEL
LIN {X 0,Y 515.224,Z 691.44,A -85,B 0,C 180,E1 4847.221,E2 4847.221} C_VEL
LIN {X 0,Y 515.017,Z 691.44,A -85,B 0,C 180,E1 4855.757,E2 4855.757} C_VEL
LIN {X 0,Y 515.197,Z 691.44,A -85,B 0,C 180,E1 4862.512,E2 4862.512} C_VEL
LIN {X 0,Y 514.764,Z 691.44,A -85,B 0,C 180,E1 4871.025,E2 4871.025} C_VEL
LIN {X 0,Y 514.537,Z 691.44,A -85,B 0,C 180,E1 4879.801,E2 4879.801} C_VEL
LIN {X 0,Y 514.383,Z 691.44,A -85,B 0,C 180,E1 4889.5,E2 4889.5} C_VEL
LIN {X 0,Y 514.294,Z 691.44,A -85,B 0,C 180,E1 4899.341,E2 4899.341} C_VEL
LIN {X 0,Y 514.245,Z 691.44,A -85,B 0,C 180,E1 4900.845,E2 4900.845} C_VEL
LIN {X 0,Y 506.176,Z 691.44,A -85,B 0,C 180,E1 4904.723,E2 4904.723} C_VEL
LIN {X 0,Y 506.528,Z 692.631,A -85,B 0,C 180,E1 4908.343,E2 4908.343} C_VEL
LIN {X 0,Y 526.819,Z 733.741,A -85,B 0,C 180,E1 4910.964,E2 4910.964} C_VEL
LIN {X 0,Y 524.166,Z 798.493,A -85,B 0,C 180,E1 4912.899,E2 4912.899} C_VEL
LIN {X 0,Y 519.305,Z 860.171,A -85,B 0,C 180,E1 4916.408,E2 4916.408} C_VEL
LIN {X 0,Y 513.808,Z 918.178,A -85,B 0,C 180,E1 4921.725,E2 4921.725} C_VEL
LIN {X 0,Y 509.74,Z 964.048,A -85,B 0,C 180,E1 4928.151,E2 4928.151} C_VEL
LIN {X 0,Y 507.651,Z 995.549,A -85,B 0,C 180,E1 4934.836,E2 4934.836} C_VEL
LIN {X 0,Y 507.06,Z 1014.285,A -85,B 0,C 180,E1 4941.393,E2 4941.393} C_VEL
LIN {X 0,Y 507.029,Z 1022.15,A -85,B 0,C 180,E1 4947.426,E2 4947.426} C_VEL
LIN {X 0,Y 507.043,Z 1020.769,A -85,B 0,C 180,E1 4954.29,E2 4954.29} C_VEL
LIN {X 0,Y 507.031,Z 1008.074,A -85,B 0,C 180,E1 4961.218,E2 4961.218} C_VEL
LIN {X 0,Y 508.228,Z 984.389,A -85,B 0,C 180,E1 4967.876,E2 4967.876} C_VEL
LIN {X 0,Y 511.12,Z 947.593,A -85,B 0,C 180,E1 4974.471,E2 4974.471} C_VEL
LIN {X 0,Y 515.936,Z 896.016,A -85,B 0,C 180,E1 4980.592,E2 4980.592} C_VEL
LIN {X 0,Y 521.288,Z 837.06,A -85,B 0,C 180,E1 4985.125,E2 4985.125} C_VEL
LIN {X 0,Y 525.669,Z 774.331,A -85,B 0,C 180,E1 4988.005,E2 4988.005} C_VEL
LIN {X 0,Y 525.413,Z 726.824,A -85,B 0,C 180,E1 4989.295,E2 4989.295} C_VEL
LIN {X 0,Y 506.391,Z 691.44,A -85,B 0,C 180,E1 4991.764,E2 4991.764} C_VEL
LIN {X 0,Y 506.316,Z 691.44,A -85,B 0,C 180,E1 5002.124,E2 5002.124} C_VEL
LIN {X 0,Y 506.4,Z 691.44,A -85,B 0,C 180,E1 5012.351,E2 5012.351} C_VEL
LIN {X 0,Y 506.617,Z 691.44,A -85,B 0,C 180,E1 5021.693,E2 5021.693} C_VEL
LIN {X 0,Y 506.72,Z 691.44,A -85,B 0,C 180,E1 5030.541,E2 5030.541} C_VEL
LIN {X 0,Y 507.022,Z 691.44,A -85,B 0,C 180,E1 5039.163,E2 5039.163} C_VEL
LIN {X 0,Y 507.126,Z 691.44,A -85,B 0,C 180,E1 5049.491,E2 5049.491} C_VEL
LIN {X 0,Y 506.67,Z 692.782,A -85,B 0,C 180,E1 5056.856,E2 5056.856} C_VEL
LIN {X 0,Y 525.792,Z 735.513,A -85,B 0,C 180,E1 5059.652,E2 5059.652} C_VEL
LIN {X 0,Y 521.553,Z 802.687,A -85,B 0,C 180,E1 5062.559,E2 5062.559} C_VEL
LIN {X 0,Y 516.301,Z 863.351,A -85,B 0,C 180,E1 5067.118,E2 5067.118} C_VEL
LIN {X 0,Y 511.814,Z 914.248,A -85,B 0,C 180,E1 5073.028,E2 5073.028} C_VEL
LIN {X 0,Y 509.015,Z 953.394,A -85,B 0,C 180,E1 5079.881,E2 5079.881} C_VEL
LIN {X 0,Y 507.742,Z 978.996,A -85,B 0,C 180,E1 5087.092,E2 5087.092} C_VEL
LIN {X 0,Y 507.086,Z 991.404,A -85,B 0,C 180,E1 5094.297,E2 5094.297} C_VEL
LIN {X 0,Y 506.729,Z 992.263,A -85,B 0,C 180,E1 5100.387,E2 5100.387} C_VEL
LIN {X 0,Y 507.123,Z 982.047,A -85,B 0,C 180,E1 5107.571,E2 5107.571} C_VEL
LIN {X 0,Y 507.992,Z 960.492,A -85,B 0,C 180,E1 5114.404,E2 5114.404} C_VEL
LIN {X 0,Y 510.445,Z 925.421,A -85,B 0,C 180,E1 5121.236,E2 5121.236} C_VEL
LIN {X 0,Y 514.956,Z 876.741,A -85,B 0,C 180,E1 5127.467,E2 5127.467} C_VEL
LIN {X 0,Y 520.453,Z 817.844,A -85,B 0,C 180,E1 5132.403,E2 5132.403} C_VEL
LIN {X 0,Y 525.001,Z 755.567,A -85,B 0,C 180,E1 5135.573,E2 5135.573} C_VEL
LIN {X 0,Y 524.594,Z 727.304,A -85,B 0,C 180,E1 5136.62,E2 5136.62} C_VEL
LIN {X 0,Y 507.168,Z 691.44,A -85,B 0,C 180,E1 5139.068,E2 5139.068} C_VEL
LIN {X 0,Y 506.67,Z 691.44,A -85,B 0,C 180,E1 5148.331,E2 5148.331} C_VEL
LIN {X 0,Y 506.435,Z 691.44,A -85,B 0,C 180,E1 5157.855,E2 5157.855} C_VEL
LIN {X 0,Y 506.258,Z 691.44,A -85,B 0,C 180,E1 5167.918,E2 5167.918} C_VEL
LIN {X 0,Y 506.349,Z 691.44,A -85,B 0,C 180,E1 5177.582,E2 5177.582} C_VEL
LIN {X 0,Y 506.334,Z 691.44,A -85,B 0,C 180,E1 5188.35,E2 5188.35} C_VEL
LIN {X 0,Y 506.288,Z 691.44,A -85,B 0,C 180,E1 5196.115,E2 5196.115} C_VEL
LIN {X 0,Y 507.233,Z 691.44,A -85,B 0,C 180,E1 5206.503,E2 5206.503} C_VEL
LIN {X 0,Y 507.018,Z 691.44,A -85,B 0,C 180,E1 5215.69,E2 5215.69} C_VEL
LIN {X 0,Y 507.196,Z 691.44,A -85,B 0,C 180,E1 5222.552,E2 5222.552} C_VEL
LIN {X 0,Y 506.738,Z 691.44,A -85,B 0,C 180,E1 5231.202,E2 5231.202} C_VEL
LIN {X 0,Y 506.547,Z 691.44,A -85,B 0,C 180,E1 5240.127,E2 5240.127} C_VEL
LIN {X 0,Y 506.394,Z 691.44,A -85,B 0,C 180,E1 5249.605,E2 5249.605} C_VEL
LIN {X 0,Y 506.249,Z 691.44,A -85,B 0,C 180,E1 5260.144,E2 5260.144} C_VEL
LIN {X 0,Y 506.176,Z 691.44,A -85,B 0,C 180,E1 5264.723,E2 5264.723} C_VEL
LIN {X 0,Y 498.323,Z 691.44,A -85,B 0,C 180,E1 5267.309,E2 5267.309} C_VEL
LIN {X 0,Y 520.584,Z 736.989,A -85,B 0,C 180,E1 5270.473,E2 5270.473} C_VEL
LIN {X 0,Y 517.605,Z 800.48,A -85,B 0,C 180,E1 5272.441,E2 5272.441} C_VEL
LIN {X 0,Y 512.162,Z 863.244,A -85,B 0,C 180,E1 5276.132,E2 5276.132} C_VEL
LIN {X 0,Y 506.439,Z 918.768,A -85,B 0,C 180,E1 5281.35,E2 5281.35} C_VEL
LIN {X 0,Y 501.921,Z 965.375,A -85,B 0,C 180,E1 5288.026,E2 5288.026} C_VEL
LIN {X 0,Y 499.604,Z 997.102,A -85,B 0,C 180,E1 5295.036,E2 5295.036} C_VEL
LIN {X 0,Y 499.038,Z 1014.783,A -85,B 0,C 180,E1 5301.516,E2 5301.516} C_VEL
LIN {X 0,Y 499.035,Z 1022.149,A -85,B 0,C 180,E1 5307.385,E2 5307.385} C_VEL
LIN {X 0,Y 499.037,Z 1020.769,A -85,B 0,C 180,E1 5314.359,E2 5314.359} C_VEL
LIN {X 0,Y 499.079,Z 1008.075,A -85,B 0,C 180,E1 5321.399,E2 5321.399} C_VEL
LIN {X 0,Y 500.417,Z 984.262,A -85,B 0,C 180,E1 5328.194,E2 5328.194} C_VEL
LIN {X 0,Y 503.596,Z 946.845,A -85,B 0,C 180,E1 5334.972,E2 5334.972} C_VEL
LIN {X 0,Y 508.849,Z 895.496,A -85,B 0,C 180,E1 5341.121,E2 5341.121} C_VEL
LIN {X 0,Y 514.77,Z 835.377,A -85,B 0,C 180,E1 5345.751,E2 5345.751} C_VEL
LIN {X 0,Y 519.374,Z 773.53,A -85,B 0,C 180,E1 5348.581,E2 5348.581} C_VEL
LIN {X 0,Y 519.345,Z 730.343,A -85,B 0,C 180,E1 5349.777,E2 5349.777} C_VEL
LIN {X 0,Y 498.339,Z 691.44,A -85,B 0,C 180,E1 5352.565,E2 5352.565} C_VEL
LIN {X 0,Y 498.199,Z 691.44,A -85,B 0,C 180,E1 5361.394,E2 5361.394} C_VEL
LIN {X 0,Y 498.374,Z 691.44,A -85,B 0,C 180,E1 5371.867,E2 5371.867} C_VEL
LIN {X 0,Y 498.639,Z 691.44,A -85,B 0,C 180,E1 5381.389,E2 5381.389} C_VEL
LIN {X 0,Y 498.721,Z 691.44,A -85,B 0,C 180,E1 5390.388,E2 5390.388} C_VEL
LIN {X 0,Y 499.016,Z 691.44,A -85,B 0,C 180,E1 5399.149,E2 5399.149} C_VEL
LIN {X 0,Y 499.078,Z 691.44,A -85,B 0,C 180,E1 5409.646,E2 5409.646} C_VEL
LIN {X 0,Y 498.878,Z 693.235,A -85,B 0,C 180,E1 5416.096,E2 5416.096} C_VEL
LIN {X 0,Y 519.407,Z 738.033,A -85,B 0,C 180,E1 5419.182,E2 5419.182} C_VEL
LIN {X 0,Y 514.774,Z 804.384,A -85,B 0,C 180,E1 5422.132,E2 5422.132} C_VEL
LIN {X 0,Y 509.133,Z 864.188,A -85,B 0,C 180,E1 5426.723,E2 5426.723} C_VEL
LIN {X 0,Y 504.166,Z 915.489,A -85,B 0,C 180,E1 5432.806,E2 5432.806} C_VEL
LIN {X 0,Y 501.05,Z 955.237,A -85,B 0,C 180,E1 5440.009,E2 5440.009} C_VEL
LIN {X 0,Y 499.497,Z 980.662,A -85,B 0,C 180,E1 5447.568,E2 5447.568} C_VEL
LIN {X 0,Y 499.039,Z 990.919,A -85,B 0,C 180,E1 5453.709,E2 5453.709} C_VEL
LIN {X 0,Y 498.728,Z 992.409,A -85,B 0,C 180,E1 5460.155,E2 5460.155} C_VEL
LIN {X 0,Y 499.223,Z 983.206,A -85,B 0,C 180,E1 5467.196,E2 5467.196} C_VEL
LIN {X 0,Y 500.094,Z 962.53,A -85,B 0,C 180,E1 5474.151,E2 5474.151} C_VEL
LIN {X 0,Y 502.658,Z 927.194,A -85,B 0,C 180,E1 5481.318,E2 5481.318} C_VEL
LIN {X 0,Y 507.609,Z 878.117,A -85,B 0,C 180,E1 5487.784,E2 5487.784} C_VEL
LIN {X 0,Y 513.459,Z 820.283,A -85,B 0,C 180,E1 5492.754,E2 5492.754} C_VEL
LIN {X 0,Y 518.496,Z 757.167,A -85,B 0,C 180,E1 5496.059,E2 5496.059} C_VEL
LIN {X 0,Y 518.264,Z 730.317,A -85,B 0,C 180,E1 5497.086,E2 5497.086} C_VEL
LIN {X 0,Y 498.973,Z 691.44,A -85,B 0,C 180,E1 5500.028,E2 5500.028} C_VEL
LIN {X 0,Y 498.653,Z 691.44,A -85,B 0,C 180,E1 5508.637,E2 5508.637} C_VEL
LIN {X 0,Y 498.416,Z 691.44,A -85,B 0,C 180,E1 5518.162,E2 5518.162} C_VEL
LIN {X 0,Y 498.189,Z 691.44,A -85,B 0,C 180,E1 5528.645,E2 5528.645} C_VEL
LIN {X 0,Y 498.236,Z 691.44,A -85,B 0,C 180,E1 5538.268,E2 5538.268} C_VEL
LIN {X 0,Y 498.258,Z 691.44,A -85,B 0,C 180,E1 5547.776,E2 5547.776} C_VEL
LIN {X 0,Y 498.311,Z 691.44,A -85,B 0,C 180,E1 5555.708,E2 5555.708} C_VEL
LIN {X 0,Y 499.22,Z 691.44,A -85,B 0,C 180,E1 5565.008,E2 5565.008} C_VEL
LIN {X 0,Y 499.018,Z 691.44,A -85,B 0,C 180,E1 5575.621,E2 5575.621} C_VEL
LIN {X 0,Y 499.177,Z 691.44,A -85,B 0,C 180,E1 5582.593,E2 5582.593} C_VEL
LIN {X 0,Y 498.714,Z 691.44,A -85,B 0,C 180,E1 5591.385,E2 5591.385} C_VEL
LIN {X 0,Y 498.531,Z 691.44,A -85,B 0,C 180,E1 5600.465,E2 5600.465} C_VEL
LIN {X 0,Y 498.372,Z 691.44,A -85,B 0,C 180,E1 5610.13,E2 5610.13} C_VEL
LIN {X 0,Y 498.154,Z 691.44,A -85,B 0,C 180,E1 5620.879,E2 5620.879} C_VEL
LIN {X 0,Y 498.323,Z 691.44,A -85,B 0,C 180,E1 5627.309,E2 5627.309} C_VEL
LIN {X 0,Y 503.053,Z 701.493,A -85,B 0,C 180,E1 5628.166,E2 5628.166} C_VEL
LIN {X 0,Y 506.903,Z 722.832,A -85,B 0,C 180,E1 5628.936,E2 5628.936} C_VEL
LIN {X 0,Y 514.312,Z 740.934,A -85,B 0,C 180,E1 5629.992,E2 5629.992} C_VEL
LIN {X 0,Y 510.898,Z 804.637,A -85,B 0,C 180,E1 5632.077,E2 5632.077} C_VEL
LIN {X 0,Y 504.896,Z 867.521,A -85,B 0,C 180,E1 5635.939,E2 5635.939} C_VEL
LIN {X 0,Y 498.69,Z 922.606,A -85,B 0,C 180,E1 5641.36,E2 5641.36} C_VEL
LIN {X 0,Y 494.108,Z 966.67,A -85,B 0,C 180,E1 5647.898,E2 5647.898} C_VEL
LIN {X 0,Y 491.729,Z 997.103,A -85,B 0,C 180,E1 5654.791,E2 5654.791} C_VEL
LIN {X 0,Y 491.067,Z 1014.818,A -85,B 0,C 180,E1 5661.397,E2 5661.397} C_VEL
LIN {X 0,Y 491.044,Z 1022.149,A -85,B 0,C 180,E1 5667.342,E2 5667.342} C_VEL
LIN {X 0,Y 491.048,Z 1020.768,A -85,B 0,C 180,E1 5674.43,E2 5674.43} C_VEL
LIN {X 0,Y 491.135,Z 1008.075,A -85,B 0,C 180,E1 5681.586,E2 5681.586} C_VEL
LIN {X 0,Y 492.613,Z 984.104,A -85,B 0,C 180,E1 5688.531,E2 5688.531} C_VEL
LIN {X 0,Y 496.143,Z 946.16,A -85,B 0,C 180,E1 5695.476,E2 5695.476} C_VEL
LIN {X 0,Y 501.868,Z 894.638,A -85,B 0,C 180,E1 5701.694,E2 5701.694} C_VEL
LIN {X 0,Y 508.282,Z 834.432,A -85,B 0,C 180,E1 5706.345,E2 5706.345} C_VEL
LIN {X 0,Y 513.131,Z 772.522,A -85,B 0,C 180,E1 5709.169,E2 5709.169} C_VEL
LIN {X 0,Y 513.028,Z 733.377,A -85,B 0,C 180,E1 5710.276,E2 5710.276} C_VEL
LIN {X 0,Y 490.282,Z 691.44,A -85,B 0,C 180,E1 5713.376,E2 5713.376} C_VEL
LIN {X 0,Y 490.145,Z 691.44,A -85,B 0,C 180,E1 5722.897,E2 5722.897} C_VEL
LIN {X 0,Y 490.256,Z 691.44,A -85,B 0,C 180,E1 5733.36,E2 5733.36} C_VEL
LIN {X 0,Y 490.568,Z 691.44,A -85,B 0,C 180,E1 5742.935,E2 5742.935} C_VEL
LIN {X 0,Y 490.909,Z 691.44,A -85,B 0,C 180,E1 5752.026,E2 5752.026} C_VEL
LIN {X 0,Y 491.181,Z 691.44,A -85,B 0,C 180,E1 5762.676,E2 5762.676} C_VEL
LIN {X 0,Y 490.751,Z 691.44,A -85,B 0,C 180,E1 5771.614,E2 5771.614} C_VEL
LIN {X 0,Y 490.833,Z 692.535,A -85,B 0,C 180,E1 5775.254,E2 5775.254} C_VEL
LIN {X 0,Y 512.991,Z 741.362,A -85,B 0,C 180,E1 5778.727,E2 5778.727} C_VEL
LIN {X 0,Y 507.972,Z 806.807,A -85,B 0,C 180,E1 5781.738,E2 5781.738} C_VEL
LIN {X 0,Y 501.76,Z 866.827,A -85,B 0,C 180,E1 5786.493,E2 5786.493} C_VEL
LIN {X 0,Y 496.475,Z 917.301,A -85,B 0,C 180,E1 5792.666,E2 5792.666} C_VEL
LIN {X 0,Y 493.144,Z 956.235,A -85,B 0,C 180,E1 5799.946,E2 5799.946} C_VEL
LIN {X 0,Y 491.341,Z 981.695,A -85,B 0,C 180,E1 5807.862,E2 5807.862} C_VEL
LIN {X 0,Y 490.824,Z 992.077,A -85,B 0,C 180,E1 5815.111,E2 5815.111} C_VEL
LIN {X 0,Y 490.765,Z 991.33,A -85,B 0,C 180,E1 5821.817,E2 5821.817} C_VEL
LIN {X 0,Y 491.104,Z 980.762,A -85,B 0,C 180,E1 5828.48,E2 5828.48} C_VEL
LIN {X 0,Y 492.302,Z 958.279,A -85,B 0,C 180,E1 5835.513,E2 5835.513} C_VEL
LIN {X 0,Y 495.476,Z 922.138,A -85,B 0,C 180,E1 5842.522,E2 5842.522} C_VEL
LIN {X 0,Y 501.129,Z 871.691,A -85,B 0,C 180,E1 5848.938,E2 5848.938} C_VEL
LIN {X 0,Y 507.409,Z 813.26,A -85,B 0,C 180,E1 5853.752,E2 5853.752} C_VEL
LIN {X 0,Y 512.538,Z 752.428,A -85,B 0,C 180,E1 5856.79,E2 5856.79} C_VEL
LIN {X 0,Y 511.855,Z 733.413,A -85,B 0,C 180,E1 5857.568,E2 5857.568} C_VEL
LIN {X 0,Y 490.845,Z 691.44,A -85,B 0,C 180,E1 5860.917,E2 5860.917} C_VEL
LIN {X 0,Y 490.59,Z 691.44,A -85,B 0,C 180,E1 5870.84,E2 5870.84} C_VEL
LIN {X 0,Y 490.347,Z 691.44,A -85,B 0,C 180,E1 5880.709,E2 5880.709} C_VEL
LIN {X 0,Y 490.178,Z 691.44,A -85,B 0,C 180,E1 5890.651,E2 5890.651} C_VEL
LIN {X 0,Y 490.011,Z 691.44,A -85,B 0,C 180,E1 5900.573,E2 5900.573} C_VEL
LIN {X 0,Y 490.212,Z 691.44,A -85,B 0,C 180,E1 5909.267,E2 5909.267} C_VEL
LIN {X 0,Y 490.067,Z 691.44,A -85,B 0,C 180,E1 5917.21,E2 5917.21} C_VEL
LIN {X 0,Y 491.231,Z 691.44,A -85,B 0,C 180,E1 5926.696,E2 5926.696} C_VEL
LIN {X 0,Y 491.016,Z 691.44,A -85,B 0,C 180,E1 5935.549,E2 5935.549} C_VEL
LIN {X 0,Y 491.177,Z 691.44,A -85,B 0,C 180,E1 5942.635,E2 5942.635} C_VEL
LIN {X 0,Y 490.694,Z 691.44,A -85,B 0,C 180,E1 5951.573,E2 5951.573} C_VEL
LIN {X 0,Y 490.537,Z 691.44,A -85,B 0,C 180,E1 5960.814,E2 5960.814} C_VEL
LIN {X 0,Y 490.269,Z 691.44,A -85,B 0,C 180,E1 5970.681,E2 5970.681} C_VEL
LIN {X 0,Y 490.128,Z 691.44,A -85,B 0,C 180,E1 5980.658,E2 5980.658} C_VEL
LIN {X 0,Y 490.334,Z 692.581,A -85,B 0,C 180,E1 5986.687,E2 5986.687} C_VEL
LIN {X 0,Y 506.903,Z 722.832,A -85,B 0,C 180,E1 5988.936,E2 5988.936} C_VEL
LIN {X 0,Y 509.158,Z 739.622,A -85,B 0,C 180,E1 5989.491,E2 5989.491} C_VEL
LIN {X 0,Y 507.39,Z 757.939,A -85,B 0,C 180,E1 5989.818,E2 5989.818} C_VEL
LIN {X 0,Y 502.899,Z 822.143,A -85,B 0,C 180,E1 5992.398,E2 5992.398} C_VEL
LIN {X 0,Y 496.366,Z 882.971,A -85,B 0,C 180,E1 5996.715,E2 5996.715} C_VEL
LIN {X 0,Y 489.658,Z 937.92,A -85,B 0,C 180,E1 6002.901,E2 6002.901} C_VEL
LIN {X 0,Y 485.361,Z 979.517,A -85,B 0,C 180,E1 6010.135,E2 6010.135} C_VEL
LIN {X 0,Y 483.634,Z 1006.913,A -85,B 0,C 180,E1 6017.771,E2 6017.771} C_VEL
LIN {X 0,Y 483.465,Z 1020.766,A -85,B 0,C 180,E1 6025.498,E2 6025.498} C_VEL
LIN {X 0,Y 483.25,Z 1022.15,A -85,B 0,C 180,E1 6032.699,E2 6032.699} C_VEL
LIN {X 0,Y 483.14,Z 1012.358,A -85,B 0,C 180,E1 6039.948,E2 6039.948} C_VEL
LIN {X 0,Y 484.368,Z 990.344,A -85,B 0,C 180,E1 6047.316,E2 6047.316} C_VEL
LIN {X 0,Y 487.624,Z 955.569,A -85,B 0,C 180,E1 6054.407,E2 6054.407} C_VEL
LIN {X 0,Y 493.491,Z 906.195,A -85,B 0,C 180,E1 6061.003,E2 6061.003} C_VEL
LIN {X 0,Y 500.382,Z 847.397,A -85,B 0,C 180,E1 6066.066,E2 6066.066} C_VEL
LIN {X 0,Y 505.84,Z 785.51,A -85,B 0,C 180,E1 6069.274,E2 6069.274} C_VEL
LIN {X 0,Y 506.778,Z 736.733,A -85,B 0,C 180,E1 6070.778,E2 6070.778} C_VEL
LIN {X 0,Y 482.245,Z 691.44,A -85,B 0,C 180,E1 6074.318,E2 6074.318} C_VEL
LIN {X 0,Y 482.05,Z 691.44,A -85,B 0,C 180,E1 6084.415,E2 6084.415} C_VEL
LIN {X 0,Y 482.213,Z 691.44,A -85,B 0,C 180,E1 6093.756,E2 6093.756} C_VEL
LIN {X 0,Y 482.575,Z 691.44,A -85,B 0,C 180,E1 6103.566,E2 6103.566} C_VEL
LIN {X 0,Y 483.189,Z 691.44,A -85,B 0,C 180,E1 6113.711,E2 6113.711} C_VEL
LIN {X 0,Y 483.162,Z 691.44,A -85,B 0,C 180,E1 6122.721,E2 6122.721} C_VEL
LIN {X 0,Y 482.767,Z 691.44,A -85,B 0,C 180,E1 6131.809,E2 6131.809} C_VEL
LIN {X 0,Y 482.909,Z 692.897,A -85,B 0,C 180,E1 6134.404,E2 6134.404} C_VEL
LIN {X 0,Y 506.604,Z 744.763,A -85,B 0,C 180,E1 6138.267,E2 6138.267} C_VEL
LIN {X 0,Y 501.03,Z 810.183,A -85,B 0,C 180,E1 6141.403,E2 6141.403} C_VEL
LIN {X 0,Y 494.303,Z 869.961,A -85,B 0,C 180,E1 6146.302,E2 6146.302} C_VEL
LIN {X 0,Y 488.727,Z 919.182,A -85,B 0,C 180,E1 6152.544,E2 6152.544} C_VEL
LIN {X 0,Y 485.193,Z 957.64,A -85,B 0,C 180,E1 6159.977,E2 6159.977} C_VEL
LIN {X 0,Y 483.48,Z 981.404,A -85,B 0,C 180,E1 6167.558,E2 6167.558} C_VEL
LIN {X 0,Y 482.849,Z 991.667,A -85,B 0,C 180,E1 6174.448,E2 6174.448} C_VEL
LIN {X 0,Y 482.636,Z 992.087,A -85,B 0,C 180,E1 6180.832,E2 6180.832} C_VEL
LIN {X 0,Y 483.146,Z 982.303,A -85,B 0,C 180,E1 6187.933,E2 6187.933} C_VEL
LIN {X 0,Y 484.228,Z 961.873,A -85,B 0,C 180,E1 6194.873,E2 6194.873} C_VEL
LIN {X 0,Y 487.32,Z 928.07,A -85,B 0,C 180,E1 6201.945,E2 6201.945} C_VEL
LIN {X 0,Y 493.044,Z 879.758,A -85,B 0,C 180,E1 6208.569,E2 6208.569} C_VEL
LIN {X 0,Y 499.852,Z 822.088,A -85,B 0,C 180,E1 6213.7,E2 6213.7} C_VEL
LIN {X 0,Y 505.736,Z 759.022,A -85,B 0,C 180,E1 6217.115,E2 6217.115} C_VEL
LIN {X 0,Y 505.411,Z 736.118,A -85,B 0,C 180,E1 6218.075,E2 6218.075} C_VEL
LIN {X 0,Y 482.763,Z 691.44,A -85,B 0,C 180,E1 6221.791,E2 6221.791} C_VEL
LIN {X 0,Y 482.557,Z 691.44,A -85,B 0,C 180,E1 6231.894,E2 6231.894} C_VEL
LIN {X 0,Y 482.302,Z 691.44,A -85,B 0,C 180,E1 6241.278,E2 6241.278} C_VEL
LIN {X 0,Y 482.167,Z 691.44,A -85,B 0,C 180,E1 6250.184,E2 6250.184} C_VEL
LIN {X 0,Y 482.047,Z 691.44,A -85,B 0,C 180,E1 6259.79,E2 6259.79} C_VEL
LIN {X 0,Y 482.185,Z 691.44,A -85,B 0,C 180,E1 6269.943,E2 6269.943} C_VEL
LIN {X 0,Y 481.973,Z 691.44,A -85,B 0,C 180,E1 6278.754,E2 6278.754} C_VEL
LIN {X 0,Y 483.19,Z 691.44,A -85,B 0,C 180,E1 6286.357,E2 6286.357} C_VEL
LIN {X 0,Y 483.013,Z 691.44,A -85,B 0,C 180,E1 6295.475,E2 6295.475} C_VEL
LIN {X 0,Y 483.158,Z 691.44,A -85,B 0,C 180,E1 6302.679,E2 6302.679} C_VEL
LIN {X 0,Y 482.707,Z 691.44,A -85,B 0,C 180,E1 6311.767,E2 6311.767} C_VEL
LIN {X 0,Y 482.491,Z 691.44,A -85,B 0,C 180,E1 6321.892,E2 6321.892} C_VEL
LIN {X 0,Y 482.217,Z 691.44,A -85,B 0,C 180,E1 6331.251,E2 6331.251} C_VEL
LIN {X 0,Y 482.113,Z 691.44,A -85,B 0,C 180,E1 6340.149,E2 6340.149} C_VEL
LIN {X 0,Y 482.36,Z 693.043,A -85,B 0,C 180,E1 6345.824,E2 6345.824} C_VEL
LIN {X 0,Y 508.105,Z 741.648,A -85,B 0,C 180,E1 6349.436,E2 6349.436} C_VEL
LIN {X 0,Y 507.39,Z 757.939,A -85,B 0,C 180,E1 6349.818,E2 6349.818} C_VEL
LIN {X 0,Y 498.908,Z 791.919,A -85,B 0,C 180,E1 6350.394,E2 6350.394} C_VEL
LIN {X 0,Y 492.597,Z 856.868,A -85,B 0,C 180,E1 6354.036,E2 6354.036} C_VEL
LIN {X 0,Y 485.315,Z 914.927,A -85,B 0,C 180,E1 6359.494,E2 6359.494} C_VEL
LIN {X 0,Y 479.566,Z 961.96,A -85,B 0,C 180,E1 6366.311,E2 6366.311} C_VEL
LIN {X 0,Y 476.282,Z 995.552,A -85,B 0,C 180,E1 6373.81,E2 6373.81} C_VEL
LIN {X 0,Y 475.236,Z 1014.284,A -85,B 0,C 180,E1 6380.812,E2 6380.812} C_VEL
LIN {X 0,Y 475.083,Z 1022.148,A -85,B 0,C 180,E1 6387.253,E2 6387.253} C_VEL
LIN {X 0,Y 475.043,Z 1020.768,A -85,B 0,C 180,E1 6394.58,E2 6394.58} C_VEL
LIN {X 0,Y 475.263,Z 1008.074,A -85,B 0,C 180,E1 6401.978,E2 6401.978} C_VEL
LIN {X 0,Y 477.257,Z 982.656,A -85,B 0,C 180,E1 6409.504,E2 6409.504} C_VEL
LIN {X 0,Y 481.931,Z 941.661,A -85,B 0,C 180,E1 6416.992,E2 6416.992} C_VEL
LIN {X 0,Y 488.487,Z 889.697,A -85,B 0,C 180,E1 6423.187,E2 6423.187} C_VEL
LIN {X 0,Y 495.463,Z 830.897,A -85,B 0,C 180,E1 6427.658,E2 6427.658} C_VEL
LIN {X 0,Y 500.779,Z 767.78,A -85,B 0,C 180,E1 6430.431,E2 6430.431} C_VEL
LIN {X 0,Y 500.316,Z 739.399,A -85,B 0,C 180,E1 6431.331,E2 6431.331} C_VEL
LIN {X 0,Y 474.18,Z 691.44,A -85,B 0,C 180,E1 6435.142,E2 6435.142} C_VEL
LIN {X 0,Y 474.01,Z 691.44,A -85,B 0,C 180,E1 6444.726,E2 6444.726} C_VEL
LIN {X 0,Y 474.193,Z 691.44,A -85,B 0,C 180,E1 6454.433,E2 6454.433} C_VEL
LIN {X 0,Y 474.621,Z 691.44,A -85,B 0,C 180,E1 6464.255,E2 6464.255} C_VEL
LIN {X 0,Y 475.154,Z 691.44,A -85,B 0,C 180,E1 6473.605,E2 6473.605} C_VEL
LIN {X 0,Y 475.165,Z 691.44,A -85,B 0,C 180,E1 6482.766,E2 6482.766} C_VEL
LIN {X 0,Y 474.71,Z 691.44,A -85,B 0,C 180,E1 6492.83,E2 6492.83} C_VEL
LIN {X 0,Y 475.227,Z 694.099,A -85,B 0,C 180,E1 6493.556,E2 6493.556} C_VEL
LIN {X 0,Y 500.357,Z 745.291,A -85,B 0,C 180,E1 6497.698,E2 6497.698} C_VEL
LIN {X 0,Y 494.434,Z 810.906,A -85,B 0,C 180,E1 6500.882,E2 6500.882} C_VEL
LIN {X 0,Y 487.237,Z 870.411,A -85,B 0,C 180,E1 6505.838,E2 6505.838} C_VEL
LIN {X 0,Y 481.063,Z 920.562,A -85,B 0,C 180,E1 6512.34,E2 6512.34} C_VEL
LIN {X 0,Y 477.352,Z 957.868,A -85,B 0,C 180,E1 6519.727,E2 6519.727} C_VEL
LIN {X 0,Y 475.416,Z 982.13,A -85,B 0,C 180,E1 6527.728,E2 6527.728} C_VEL
LIN {X 0,Y 474.841,Z 991.834,A -85,B 0,C 180,E1 6534.602,E2 6534.602} C_VEL
LIN {X 0,Y 474.769,Z 990.954,A -85,B 0,C 180,E1 6542.388,E2 6542.388} C_VEL
LIN {X 0,Y 475.367,Z 978.119,A -85,B 0,C 180,E1 6549.926,E2 6549.926} C_VEL
LIN {X 0,Y 477.462,Z 951.983,A -85,B 0,C 180,E1 6557.612,E2 6557.612} C_VEL
LIN {X 0,Y 482.052,Z 910.733,A -85,B 0,C 180,E1 6565.084,E2 6565.084} C_VEL
LIN {X 0,Y 488.834,Z 857.644,A -85,B 0,C 180,E1 6571.335,E2 6571.335} C_VEL
LIN {X 0,Y 496.057,Z 796.11,A -85,B 0,C 180,E1 6575.927,E2 6575.927} C_VEL
LIN {X 0,Y 499.317,Z 739.702,A -85,B 0,C 180,E1 6578.53,E2 6578.53} C_VEL
LIN {X 0,Y 474.698,Z 691.44,A -85,B 0,C 180,E1 6582.786,E2 6582.786} C_VEL
LIN {X 0,Y 474.552,Z 691.44,A -85,B 0,C 180,E1 6591.579,E2 6591.579} C_VEL
LIN {X 0,Y 474.198,Z 691.44,A -85,B 0,C 180,E1 6601.978,E2 6601.978} C_VEL
LIN {X 0,Y 474.081,Z 691.44,A -85,B 0,C 180,E1 6611.197,E2 6611.197} C_VEL
LIN {X 0,Y 473.98,Z 691.44,A -85,B 0,C 180,E1 6621.349,E2 6621.349} C_VEL
LIN {X 0,Y 474.195,Z 691.44,A -85,B 0,C 180,E1 6631.656,E2 6631.656} C_VEL
LIN {X 0,Y 474.532,Z 691.44,A -85,B 0,C 180,E1 6642.295,E2 6642.295} C_VEL
LIN {X 0,Y 474.779,Z 691.44,A -85,B 0,C 180,E1 6649.856,E2 6649.856} C_VEL
LIN {X 0,Y 475.032,Z 691.44,A -85,B 0,C 180,E1 6659.064,E2 6659.064} C_VEL
LIN {X 0,Y 475.054,Z 691.44,A -85,B 0,C 180,E1 6668.242,E2 6668.242} C_VEL
LIN {X 0,Y 474.621,Z 691.44,A -85,B 0,C 180,E1 6677.657,E2 6677.657} C_VEL
LIN {X 0,Y 474.218,Z 691.44,A -85,B 0,C 180,E1 6687.616,E2 6687.616} C_VEL
LIN {X 0,Y 474.051,Z 691.44,A -85,B 0,C 180,E1 6698.34,E2 6698.34} C_VEL
LIN {X 0,Y 474.281,Z 693.047,A -85,B 0,C 180,E1 6704.899,E2 6704.899} C_VEL
LIN {X 0,Y 501.801,Z 744.869,A -85,B 0,C 180,E1 6708.919,E2 6708.919} C_VEL
LIN {X 0,Y 498.908,Z 791.919,A -85,B 0,C 180,E1 6710.394,E2 6710.394} C_VEL
LIN {X 0,Y 489.572,Z 824.959,A -85,B 0,C 180,E1 6711.436,E2 6711.436} C_VEL
LIN {X 0,Y 482.205,Z 885.76,A -85,B 0,C 180,E1 6715.904,E2 6715.904} C_VEL
LIN {X 0,Y 474.779,Z 938.762,A -85,B 0,C 180,E1 6722.104,E2 6722.104} C_VEL
LIN {X 0,Y 469.8,Z 979.292,A -85,B 0,C 180,E1 6729.398,E2 6729.398} C_VEL
LIN {X 0,Y 467.574,Z 1006.507,A -85,B 0,C 180,E1 6737.176,E2 6737.176} C_VEL
LIN {X 0,Y 467.427,Z 1020.766,A -85,B 0,C 180,E1 6745.343,E2 6745.343} C_VEL
LIN {X 0,Y 467.237,Z 1022.149,A -85,B 0,C 180,E1 6752.792,E2 6752.792} C_VEL
LIN {X 0,Y 467.133,Z 1012.358,A -85,B 0,C 180,E1 6760.292,E2 6760.292} C_VEL
LIN {X 0,Y 468.531,Z 991.947,A -85,B 0,C 180,E1 6767.474,E2 6767.474} C_VEL
LIN {X 0,Y 472.325,Z 957.347,A -85,B 0,C 180,E1 6774.942,E2 6774.942} C_VEL
LIN {X 0,Y 479.013,Z 908.51,A -85,B 0,C 180,E1 6781.76,E2 6781.76} C_VEL
LIN {X 0,Y 486.363,Z 852.777,A -85,B 0,C 180,E1 6786.776,E2 6786.776} C_VEL
LIN {X 0,Y 492.861,Z 788.841,A -85,B 0,C 180,E1 6790.286,E2 6790.286} C_VEL
LIN {X 0,Y 494.389,Z 743.066,A -85,B 0,C 180,E1 6791.823,E2 6791.823} C_VEL
LIN {X 0,Y 466.063,Z 691.44,A -85,B 0,C 180,E1 6796.21,E2 6796.21} C_VEL
LIN {X 0,Y 466.01,Z 691.44,A -85,B 0,C 180,E1 6806.141,E2 6806.141} C_VEL
LIN {X 0,Y 466.218,Z 691.44,A -85,B 0,C 180,E1 6816.02,E2 6816.02} C_VEL
LIN {X 0,Y 466.737,Z 691.44,A -85,B 0,C 180,E1 6825.911,E2 6825.911} C_VEL
LIN {X 0,Y 467.052,Z 691.44,A -85,B 0,C 180,E1 6835.363,E2 6835.363} C_VEL
LIN {X 0,Y 467.147,Z 691.44,A -85,B 0,C 180,E1 6842.814,E2 6842.814} C_VEL
LIN {X 0,Y 466.876,Z 692.989,A -85,B 0,C 180,E1 6852.528,E2 6852.528} C_VEL
LIN {X 0,Y 493.973,Z 748.543,A -85,B 0,C 180,E1 6857.217,E2 6857.217} C_VEL
LIN {X 0,Y 487.609,Z 813.871,A -85,B 0,C 180,E1 6860.493,E2 6860.493} C_VEL
LIN {X 0,Y 480.01,Z 872.027,A -85,B 0,C 180,E1 6865.485,E2 6865.485} C_VEL
LIN {X 0,Y 473.539,Z 920.778,A -85,B 0,C 180,E1 6871.94,E2 6871.94} C_VEL
LIN {X 0,Y 469.441,Z 958.797,A -85,B 0,C 180,E1 6879.651,E2 6879.651} C_VEL
LIN {X 0,Y 467.368,Z 982.702,A -85,B 0,C 180,E1 6887.829,E2 6887.829} C_VEL
LIN {X 0,Y 466.735,Z 992.273,A -85,B 0,C 180,E1 6895.32,E2 6895.32} C_VEL
LIN {X 0,Y 466.963,Z 990.054,A -85,B 0,C 180,E1 6903.365,E2 6903.365} C_VEL
LIN {X 0,Y 468.088,Z 974.318,A -85,B 0,C 180,E1 6911.573,E2 6911.573} C_VEL
LIN {X 0,Y 470.824,Z 943.539,A -85,B 0,C 180,E1 6919.789,E2 6919.789} C_VEL
LIN {X 0,Y 476.196,Z 900.18,A -85,B 0,C 180,E1 6927.032,E2 6927.032} C_VEL
LIN {X 0,Y 483.632,Z 844.946,A -85,B 0,C 180,E1 6933.036,E2 6933.036} C_VEL
LIN {X 0,Y 490.854,Z 782.105,A -85,B 0,C 180,E1 6937.29,E2 6937.29} C_VEL
LIN {X 0,Y 492.969,Z 742.634,A -85,B 0,C 180,E1 6939.048,E2 6939.048} C_VEL
LIN {X 0,Y 466.731,Z 691.44,A -85,B 0,C 180,E1 6943.561,E2 6943.561} C_VEL
LIN {X 0,Y 466.485,Z 691.44,A -85,B 0,C 180,E1 6953.996,E2 6953.996} C_VEL
LIN {X 0,Y 466.052,Z 691.44,A -85,B 0,C 180,E1 6963.848,E2 6963.848} C_VEL
LIN {X 0,Y 466.01,Z 691.44,A -85,B 0,C 180,E1 6974.441,E2 6974.441} C_VEL
LIN {X 0,Y 466.042,Z 691.44,A -85,B 0,C 180,E1 6985.243,E2 6985.243} C_VEL
LIN {X 0,Y 466.217,Z 691.44,A -85,B 0,C 180,E1 6993.915,E2 6993.915} C_VEL
LIN {X 0,Y 467.113,Z 691.44,A -85,B 0,C 180,E1 7005.878,E2 7005.878} C_VEL
LIN {X 0,Y 467.018,Z 691.44,A -85,B 0,C 180,E1 7015.32,E2 7015.32} C_VEL
LIN {X 0,Y 467.142,Z 691.44,A -85,B 0,C 180,E1 7022.771,E2 7022.771} C_VEL
LIN {X 0,Y 466.693,Z 691.44,A -85,B 0,C 180,E1 7032.177,E2 7032.177} C_VEL
LIN {X 0,Y 466.449,Z 691.44,A -85,B 0,C 180,E1 7041.988,E2 7041.988} C_VEL
LIN {X 0,Y 466.04,Z 691.44,A -85,B 0,C 180,E1 7052.465,E2 7052.465} C_VEL
LIN {X 0,Y 465.928,Z 691.44,A -85,B 0,C 180,E1 7062.872,E2 7062.872} C_VEL
LIN {X 0,Y 466.322,Z 693.61,A -85,B 0,C 180,E1 7063.955,E2 7063.955} C_VEL
LIN {X 0,Y 495.533,Z 748.057,A -85,B 0,C 180,E1 7068.401,E2 7068.401} C_VEL
LIN {X 0,Y 490.785,Z 813.254,A -85,B 0,C 180,E1 7070.804,E2 7070.804} C_VEL
LIN {X 0,Y 489.572,Z 824.959,A -85,B 0,C 180,E1 7071.436,E2 7071.436} C_VEL
LIN {X 0,Y 479.133,Z 856.485,A -85,B 0,C 180,E1 7072.905,E2 7072.905} C_VEL
LIN {X 0,Y 471.223,Z 914.026,A -85,B 0,C 180,E1 7078.364,E2 7078.364} C_VEL
LIN {X 0,Y 464.836,Z 960.049,A -85,B 0,C 180,E1 7085.143,E2 7085.143} C_VEL
LIN {X 0,Y 460.748,Z 994.898,A -85,B 0,C 180,E1 7093.059,E2 7093.059} C_VEL
LIN {X 0,Y 459.346,Z 1014.284,A -85,B 0,C 180,E1 7100.491,E2 7100.491} C_VEL
LIN {X 0,Y 459.091,Z 1022.148,A -85,B 0,C 180,E1 7107.157,E2 7107.157} C_VEL
LIN {X 0,Y 459.058,Z 1020.768,A -85,B 0,C 180,E1 7114.74,E2 7114.74} C_VEL
LIN {X 0,Y 459.422,Z 1008.074,A -85,B 0,C 180,E1 7122.398,E2 7122.398} C_VEL
LIN {X 0,Y 462.108,Z 980.847,A -85,B 0,C 180,E1 7130.6,E2 7130.6} C_VEL
LIN {X 0,Y 467.692,Z 938.843,A -85,B 0,C 180,E1 7138.343,E2 7138.343} C_VEL
LIN {X 0,Y 474.819,Z 888.2,A -85,B 0,C 180,E1 7144.382,E2 7144.382} C_VEL
LIN {X 0,Y 482.736,Z 826.763,A -85,B 0,C 180,E1 7149.022,E2 7149.022} C_VEL
LIN {X 0,Y 488.692,Z 762.78,A -85,B 0,C 180,E1 7151.765,E2 7151.765} C_VEL
LIN {X 0,Y 487.832,Z 745.71,A -85,B 0,C 180,E1 7152.402,E2 7152.402} C_VEL
LIN {X 0,Y 457.962,Z 691.44,A -85,B 0,C 180,E1 7157.252,E2 7157.252} C_VEL
LIN {X 0,Y 458.009,Z 691.44,A -85,B 0,C 180,E1 7167.663,E2 7167.663} C_VEL
LIN {X 0,Y 458.332,Z 691.44,A -85,B 0,C 180,E1 7177.648,E2 7177.648} C_VEL
LIN {X 0,Y 458.761,Z 691.44,A -85,B 0,C 180,E1 7187.609,E2 7187.609} C_VEL
LIN {X 0,Y 458.839,Z 691.44,A -85,B 0,C 180,E1 7197.179,E2 7197.179} C_VEL
LIN {X 0,Y 458.844,Z 691.44,A -85,B 0,C 180,E1 7204.764,E2 7204.764} C_VEL
LIN {X 0,Y 458.959,Z 693.221,A -85,B 0,C 180,E1 7211.523,E2 7211.523} C_VEL
LIN {X 0,Y 487.443,Z 749.716,A -85,B 0,C 180,E1 7216.612,E2 7216.612} C_VEL
LIN {X 0,Y 481.032,Z 815.037,A -85,B 0,C 180,E1 7219.972,E2 7219.972} C_VEL
LIN {X 0,Y 472.84,Z 873.394,A -85,B 0,C 180,E1 7225.089,E2 7225.089} C_VEL
LIN {X 0,Y 465.877,Z 922.112,A -85,B 0,C 180,E1 7231.71,E2 7231.71} C_VEL
LIN {X 0,Y 461.564,Z 959.086,A -85,B 0,C 180,E1 7239.408,E2 7239.408} C_VEL
LIN {X 0,Y 459.552,Z 982.177,A -85,B 0,C 180,E1 7247.393,E2 7247.393} C_VEL
LIN {X 0,Y 458.718,Z 991.931,A -85,B 0,C 180,E1 7254.624,E2 7254.624} C_VEL
LIN {X 0,Y 458.602,Z 991.905,A -85,B 0,C 180,E1 7261.327,E2 7261.327} C_VEL
LIN {X 0,Y 459.174,Z 981.86,A -85,B 0,C 180,E1 7268.682,E2 7268.682} C_VEL
LIN {X 0,Y 460.751,Z 960.772,A -85,B 0,C 180,E1 7276.067,E2 7276.067} C_VEL
LIN {X 0,Y 464.777,Z 926.711,A -85,B 0,C 180,E1 7283.439,E2 7283.439} C_VEL
LIN {X 0,Y 472.157,Z 877.288,A -85,B 0,C 180,E1 7290.387,E2 7290.387} C_VEL
LIN {X 0,Y 480.387,Z 820.479,A -85,B 0,C 180,E1 7295.542,E2 7295.542} C_VEL
LIN {X 0,Y 487.22,Z 759.047,A -85,B 0,C 180,E1 7298.906,E2 7298.906} C_VEL
LIN {X 0,Y 485.925,Z 743.887,A -85,B 0,C 180,E1 7299.721,E2 7299.721} C_VEL
LIN {X 0,Y 458.711,Z 691.44,A -85,B 0,C 180,E1 7304.612,E2 7304.612} C_VEL
LIN {X 0,Y 458.409,Z 691.44,A -85,B 0,C 180,E1 7314.446,E2 7314.446} C_VEL
LIN {X 0,Y 458.06,Z 691.44,A -85,B 0,C 180,E1 7323.139,E2 7323.139} C_VEL
LIN {X 0,Y 457.994,Z 691.44,A -85,B 0,C 180,E1 7332.789,E2 7332.789} C_VEL
LIN {X 0,Y 457.838,Z 691.44,A -85,B 0,C 180,E1 7342.161,E2 7342.161} C_VEL
LIN {X 0,Y 458.159,Z 691.44,A -85,B 0,C 180,E1 7351.377,E2 7351.377} C_VEL
LIN {X 0,Y 458.327,Z 691.44,A -85,B 0,C 180,E1 7361.647,E2 7361.647} C_VEL
LIN {X 0,Y 458.776,Z 691.44,A -85,B 0,C 180,E1 7369.498,E2 7369.498} C_VEL
LIN {X 0,Y 459.019,Z 691.44,A -85,B 0,C 180,E1 7379.031,E2 7379.031} C_VEL
LIN {X 0,Y 459.007,Z 691.44,A -85,B 0,C 180,E1 7388.532,E2 7388.532} C_VEL
LIN {X 0,Y 458.517,Z 691.44,A -85,B 0,C 180,E1 7398.299,E2 7398.299} C_VEL
LIN {X 0,Y 458.163,Z 691.44,A -85,B 0,C 180,E1 7408.672,E2 7408.672} C_VEL
LIN {X 0,Y 457.901,Z 691.44,A -85,B 0,C 180,E1 7418.844,E2 7418.844} C_VEL
LIN {X 0,Y 458.167,Z 693.314,A -85,B 0,C 180,E1 7422.921,E2 7422.921} C_VEL
LIN {X 0,Y 489.366,Z 750.488,A -85,B 0,C 180,E1 7427.852,E2 7427.852} C_VEL
LIN {X 0,Y 484.256,Z 814.9,A -85,B 0,C 180,E1 7430.3,E2 7430.3} C_VEL
LIN {X 0,Y 479.133,Z 856.485,A -85,B 0,C 180,E1 7432.905,E2 7432.905} C_VEL
LIN {X 0,Y 468.241,Z 886.122,A -85,B 0,C 180,E1 7434.871,E2 7434.871} C_VEL
LIN {X 0,Y 460.007,Z 939.157,A -85,B 0,C 180,E1 7441.19,E2 7441.19} C_VEL
LIN {X 0,Y 454.251,Z 979.499,A -85,B 0,C 180,E1 7448.708,E2 7448.708} C_VEL
LIN {X 0,Y 451.61,Z 1006.065,A -85,B 0,C 180,E1 7456.538,E2 7456.538} C_VEL
LIN {X 0,Y 451.244,Z 1019.889,A -85,B 0,C 180,E1 7464.208,E2 7464.208} C_VEL
LIN {X 0,Y 451.211,Z 1022.149,A -85,B 0,C 180,E1 7472.891,E2 7472.891} C_VEL
LIN {X 0,Y 451.154,Z 1012.358,A -85,B 0,C 180,E1 7480.661,E2 7480.661} C_VEL
LIN {X 0,Y 452.829,Z 991.605,A -85,B 0,C 180,E1 7488.199,E2 7488.199} C_VEL
LIN {X 0,Y 457.264,Z 957.344,A -85,B 0,C 180,E1 7495.823,E2 7495.823} C_VEL
LIN {X 0,Y 464.567,Z 909.951,A -85,B 0,C 180,E1 7502.615,E2 7502.615} C_VEL
LIN {X 0,Y 473.108,Z 851.774,A -85,B 0,C 180,E1 7507.966,E2 7507.966} C_VEL
